// TwinCAT 3 PLC project PLC5236
// ProgramVersion: 3.1.4026.21
// libraries:
//   Tc2_EtherCAT, * (Beckhoff Automation GmbH)
//   Tc2_SerialCom, * (Beckhoff Automation GmbH)
//   Tc2_Standard, * (Beckhoff Automation GmbH)
//   Tc2_System, * (Beckhoff Automation GmbH)
//   Tc2_TcpIp, * (Beckhoff Automation GmbH)
//   Tc2_Utilities, * (Beckhoff Automation GmbH)
//   Tc3_Module, * (Beckhoff Automation GmbH)
//   VisuDialogs, * (System)
// project tree:
//   Data types/DATA_user/ USER.TcDUT, USER_ACTU.TcDUT, USER_GROUP.TcDUT
//   Data types/STRUCT COM TCPIP/ E_ClientSteps.TcDUT, E_DataExchaSteps.TcDUT, STRUCT_ClientConnect.TcDUT, STRUCT_LOG_TCPIP_CLIENT.TcDUT
//   Data types/STRUCTURE_STD/ STRUCT_JEV.TcDUT
//   Data types/ STRUCT_EVENT.TcDUT
//   Global Variables/ CONSTANT_COM_TCPIP_XTC.TcGVL, Global_Variables.TcGVL, Variable_Configuration.TcGVL
//   / PlcTask.TcTTO, Visualization Manager.TcVMO (not stored), VISU_TASK.TcTTO
//   POUs/Composant/AXES/ BLOCK_VARIATEUR_MOTEUR.TcPOU
//   POUs/Composant/ BLOCK_ACTUATOR.TcPOU, BLOCK_ACTUATOR2.TcPOU, BLOCK_VERRINE.TcPOU, MC_Reset_AX5000.TcPOU
//   POUs/Composant/EVAP/ BLOCK_CANON_ST10.TcPOU, BLOCK_IND_CREUSET_GENIUS.TcPOU, BLOCK_IND_CR_379_TELEMARK_V4.TcPOU, BLOCK_IND_CR_379_TELEMARK_V3.TcPOU, BLOCK_IND_CR_396_TELEMARK.TcPOU, BLOCK_SOURCE_GENIUS.TcPOU, BLOCK_SOURCE_JOULE.TcPOU, BLOCK_SWEEP_TELEMARK_PROG.TcPOU, BLOCK_TELEMARK_DIGITAL_SWEEP.TcPOU, BLOCK_TELEMARK_CHEETAH_SWEEP.TcPOU, BLOCK_XTAL.TcPOU, BLOCK_XTAL6.TcPOU
//   POUs/Composant/GAZ/ BLOCK_CONTROL_GAZ.TcPOU, BLOCK_MFC_ANA2.TcPOU, BLOCK_MFC_BKH.TcPOU, BLOCK_MFC_BROOKS_NoCoE.TcPOU, BLOCK_MFC_MKS_NoCoE.TcPOU
//   POUs/Composant/GENERATEURS/ ALIM_EFFLUVAGE.TcPOU
//   POUs/Composant/JAUGES/ BLOCK_BCG450_ANA.TcPOU, BLOCK_BCG450_ETHERCAT.TcPOU, BLOCK_CDG_ANA.TcPOU, BLOCK_CDG_ETHERCAT.TcPOU, BLOCK_ZX1_ANA.TcPOU
//   POUs/Composant/MVTS/ BLOCK_AXE_STD1.TcPOU, BLOCK_MOTEUR_ATV_ANA.TcPOU, BLOCK_MOTEUR_ATV_ETHERCAT.TcPOU, FB_WritePosBias.TcPOU, F_ReadMotorAbsPosition.TcPOU
//   POUs/Composant/POMPES/ BLOCK_PCR_CTI_OB.TcPOU, BLOCK_PPM.TcPOU, BLOCK_PPM_DEF.TcPOU, BLOCK_PTM_OBCV4.TcPOU, BLOCK_RS232_ONBOARD.TcPOU
//   POUs/Composant/POMPES/CRYO CTI/ BLOCK_RS232_ONBOARD_V4.TcPOU, Lecture_valeur.TcPOU
//   POUs/Composant/SERVITUDES/ BLOCK_CHILLER.TcPOU, BLOCK_CTA_HOT_COLD.TcPOU, BLOCK_SV4200.TcPOU
//   POUs/Composant/VANNES/ BLOCK_VVAT_3P.TcPOU, BLOCK_VVAT_650_ETHERCAT.TcPOU, BLOCK_VVAT_650_NO.TcPOU, BLOCK_VVAT_653_ETHERCAT.TcPOU
//   POUs/Composant/VERRINE/ BLOCK_BUZZER.TcPOU
//   POUs/FONCTION DE BASE/ ANALOG_INPUT.TcPOU, ANALOG_OUTPUT.TcPOU, BLOCK_CLIGNOTANT.TcPOU, BLOCK_CLIGNOTANT_V0_0.TcPOU, BLOCK_G7.TcPOU, BLOCK_OPERATION.TcPOU, BLOCK_RAMP.TcPOU, BLOCK_USER.TcPOU, IEEE754_INPUT.TcPOU, IEEE754_OUTPUT.TcPOU, LOG_EVENT.TcPOU, PRCDEF.TcPOU, SURVPRC.TcPOU, WRITE_CoE_BOOL.TcPOU, WRITE_CoE_WORD.TcPOU
//   POUs/FONCTION DE BASE/Format String/ FORMAT_FLOAT_STRING.TcPOU
//   POUs/Fonction/ETHER COM/ BLOCK_XTC3.TcPOU, BLOCK_XTC_CLIENT_EXCHANGE.TcPOU
//   POUs/Fonction/FONCTION EFFLUVAGE/ BLOCK_EFFLUVAGE.TcPOU
//   POUs/Fonction/FONCTION EVAPORATION/ BLOCK_EVAP.TcPOU, BLOCK_STEP_EMPILEMENT.TcPOU
//   POUs/Fonction/FONCTION MODEMARCHE/ BLOCK_1RUN_1QUARTZ.TcPOU, BLOCK_EXEC_PROC.TcPOU, BLOCK_INIT_MACHINE.TcPOU, BLOCK_MODE_MARCHE_V2_0.TcPOU, BLOCK_STEP_BOUCLE.TcPOU, BLOCK_STEP_EFFLUVAGE.TcPOU, BLOCK_STEP_TIMER.TcPOU, BLOCK_SYNCHRO_HORAIRE.TcPOU, BLOCK_USER_ACK.TcPOU
//   POUs/Fonction/FONCTION PS/ BLOCK_ROTATION_PS.TcPOU
//   POUs/Fonction/FONCTIONS COMPTEUR/ BLOCK_CPT_APP.TcPOU, BLOCK_CPT_INTEG.TcPOU, BLOCK_CPT_TEMPS.TcPOU
//   POUs/Fonction/FONCTIONS GAZ/ BLOCK_LIGNE_GAZ.TcPOU, BLOCK_LIGNE_GAZ_2_VANNES.TcPOU, BLOCK_LIGNE_GAZ_NO_DG.TcPOU, BLOCK_REGUL_PR_GAZ.TcPOU
//   POUs/Fonction/FONCTIONS MVTS/ BLOCK_ROTATION_CONTINUE_ATV.TcPOU
//   POUs/Fonction/FONCTIONS POMPAGE/ BLOCK_POMP_1E_PCR_PPM_ASS_ETHERCAT.TcPOU, BLOCK_POMP_1E_PCR_PPM_ASS_ETHERCAT_SINGER.TcPOU
//   POUs/Fonction/FONCTIONS PUISSANCE/ BLOCK_CPT_USURE.TcPOU, BLOCK_CPT_USURE_OLD.TcPOU
//   POUs/Fonction/FONCTIONS SERVITUDES/ BLOCK_LIGNE_REF.TcPOU, BLOCK_LIGNE_REF_FLOWTEMP.TcPOU, BLOCK_WREFCH1.TcPOU
//   POUs/Fonction/FONCTIONS UTILITAIRES/ CHECKSUM.TcPOU
//   POUs/Programme/ BLOCK_PRG_EFFLUVAGE.TcPOU, BLOCK_PRG_EVAP.TcPOU, BLOCK_PRG_GAZ.TcPOU, BLOCK_PRG_INFO_CLIENT.TcPOU, BLOCK_PRG_MOUVEMENT_PS.TcPOU, BLOCK_PRG_POMPAGE.TcPOU, BLOCK_PRG_SERVITUDES.TcPOU, BLOCK_PRG_VERRINE.TcPOU, MAIN.TcPOU, PRG_DEF_MANAGEMENT.TcPOU, PRG_SEC.TcPOU
//   TextLists/ GlobalTextList.TcGTLO, TextList_1Run_1Quartz.TcTLO, TextList_Actuator_Type.TcTLO, TextList_Basiques.TcTLO, TextList_Canne_Transfert.TcTLO, TextList_Chauffage.TcTLO, TextList_Config_Chauffage.TcTLO, TextList_Config_EFFLUVAGE.TcTLO, TextList_Config_Evap.TcTLO, TextList_Config_Gaz.TcTLO, TextList_Config_IAD.TcTLO, TextList_Config_Mouvements.TcTLO, TextList_Config_Pompage.TcTLO, TextList_CryoPump.TcTLO, TextList_Cryo_Relays_Parameters.TcTLO, TextList_EcoMode.TcTLO, TextList_Effluvage.TcTLO, TextList_Evap.TcTLO, TextList_Gaz.TcTLO, TextList_IAD.TcTLO, TextList_IC6.TcTLO, TextList_Infos.TcTLO, TextList_Moteurs.TcTLO, TextList_Navigation.TcTLO, TextList_Orders.TcTLO, TextList_Pompage.TcTLO, TextList_Position_Canne.TcTLO, TextList_Process.TcTLO, TextList_SA_Operations.TcTLO, TextList_Servitudes.TcTLO, TextList_STATE_Mode_Marche.TcTLO, TextList_Test_RP.TcTLO, TextList_Type_Etape.TcTLO, TextList_Type_Moteur.TcTLO, TextList_Users_Menu.TcTLO, TextList_Util_Defaut.TcTLO, TextList_Util_Group.TcTLO, TextList_Util_Userlist.TcTLO, TextList_VVAT_3P.TcTLO, TextList_VVAT_650_ETHERCAT.TcTLO
//   Visualizations/Config/Bandeaux/ VISU_BANDEAU_CFG.TcVIS
//   Visualizations/Config/CRYO/ VISU_CONFIG_REGEN.TcVIS
//   Visualizations/Config/ECOMODE/ VISU_CONFIG_ECOMODE.TcVIS
//   Visualizations/Config/EFFLUVAGE/ VISU_CONFIG_EFFLUV.TcVIS (excluded from build)
//   Visualizations/Config/EVAP/ VISU_CONFIG_EVAP.TcVIS
//   Visualizations/Config/GAZ/ VISU_CONFIG_GAZ.TcVIS
//   Visualizations/Config/MOUVEMENTS/ VISU_CONFIG_MOUVEMENTS.TcVIS
//   Visualizations/Config/POMPAGE/ VISU_CONFIG_POMPAGE.TcVIS
//   Visualizations/ MesImages.TcIPO (not stored)
//   Visualizations/Semi Auto/Elements/ SA_CACHE_ACTUATOR.TcVIS, SA_CACHE_ACTUATOR2.TcVIS, SA_EFFLUVAGE.TcVIS, SA_EVAP.TcVIS, SA_HEATING.TcVIS, SA_IAD.TcVIS, SA_LIGNE_GAZ_ANA_RAMPE.TcVIS, SA_LIGNE_GAZ_BROOKS_RAMPE.TcVIS, SA_LIGNE_GAZ_MKS_RAMPE.TcVIS, SA_POMP_1E_PCR_PPM.TcVIS, SA_POMP_1E_PCR_PPM_ASS.TcVIS, SA_POMP_1E_PCR_PPM_ASS_M11.TcVIS, SA_POMP_2E_PCR_PPM_ASS.TcVIS, SA_POMP_ENCEINTE.TcVIS, SA_POMP_SAS.TcVIS, SA_PS.TcVIS (excluded from build), SA_REGUL_GAZ.TcVIS, SA_ROT.TcVIS, SA_TEST_RP.TcVIS, SA_VERIN.TcVIS
//   Visualizations/Semi Auto/ VISU_SA.TcVIS
//   Visualizations/Symbole/CACHE/ SYM_CACHE.TcVIS, SYM_CACHE_ACTUATOR2.TcVIS
//   Visualizations/Symbole/Chauffage/ VISU_CHAUFF.TcVIS, VISU_CONFIG_CHAUFF.TcVIS, VISU_LAMPE.TcVIS
//   Visualizations/Symbole/DIVERS/ CHRONO.TcVIS
//   Visualizations/Symbole/Effluvage/ VISU_CONFIG_EFF.TcVIS, VISU_EFFLUVAGE.TcVIS
//   Visualizations/Symbole/EVAP/ VISU_ALIM_HT.TcVIS, VISU_ALIM_HT_S10.TcVIS, VISU_BAL_MANU.TcVIS, VISU_CANON.TcVIS, VISU_CANON_GENIUS_ETH.TcVIS, VISU_CANON_ST10.TcVIS, VISU_CONF_BAL.TcVIS, VISU_CONF_MAT.TcVIS, VISU_CREUSET_old.TcVIS, VISU_CREUSET.TcVIS, VISU_CREUSET_V3.TcVIS, VISU_CR_SW_GENIUS_ETH.TcVIS, VISU_HT_CANON_ST10.TcVIS, VISU_HT_GENIUS_ETH.TcVIS, VISU_SOURCE_EFFET_JOULE.TcVIS, VISU_SOURCE_EVAP_COTE_GENIUS_ETH.TcVIS, VISU_SOURCE_EVAP_COTE_ST10.TcVIS, VISU_SOURCE_EVAP_COTE_ST10_avec_emission.TcVIS, VISU_SWEEP_DIGITAL.TcVIS, VISU_SWEEP_CHEETAH.TcVIS, VISU_XTAL.TcVIS, VISU_XTAL6_ZOOM.TcVIS, VISU_XTAL6_PROD.TcVIS, VISU_XTAL_6.TcVIS
//   Visualizations/Symbole/GAZ/ VISU_CONFIG_LIGNE_GAZ_SEUIL.TcVIS, VISU_CONFIG_LIGNE_GAZ_SEUIL_MFC_MKS.TcVIS, VISU_CONFIG_LIGNE_GAZ_SURV.TcVIS, VISU_CONFIG_LIGNE_GAZ_SURV_MFC_MKS.TcVIS, VISU_CONFIG_REGUL_GAZ.TcVIS, VISU_LIGNE_GAZ.TcVIS, VISU_LIGNE_GAZ_ANA.TcVIS, VISU_LIGNE_GAZ_VGAUCHE.TcVIS, VISU_MFC_ANA.TcVIS, VISU_MFC_BROOKS.TcVIS, VISU_MFC_MKS.TcVIS
//   Visualizations/Symbole/IAD/ VISU_MARK3_PLUS.TcVIS, VISU_MARK3_PLUS_COTE.TcVIS
//   Visualizations/Symbole/JAUGES/ VISU_JAUGE_BCG450_V_HAUT.TcVIS, VISU_JAUGE_BCG450_V_HAUT_ETHERCAT.TcVIS, VISU_JAUGE_CDG045_ETHERCAT.TcVIS, VISU_JAUGE_PCG550_ETHERCAT.TcVIS
//   Visualizations/Symbole/MESURE/ VISU_IC6.TcVIS, VISU_XTC.TcVIS
//   Visualizations/Symbole/MODE_MARCHE/ VISU_BANDEAU.TcVIS, VISU_BLANCK_MANUEL.TcVIS, VISU_ECOMODE.TcVIS, VISU_ECOMODE_EVAP.TcVIS, VISU_EV_EXTRAIT.TcVIS, VISU_FCTS_SA.TcVIS, VISU_MODE_MARCHE.TcVIS
//   Visualizations/Symbole/MOUVEMENTS PS/AXE STD1/FCT_Part/ VISU_AXE_STD1_FCT_MANU.TcVIS, VISU_AXE_STD1_FCT_MANU_OSC.TcVIS, VISU_AXE_STD1_FCT_OP.TcVIS, VISU_AXE_STD1_FCT_OP_OSC.TcVIS, VISU_AXE_STD1_FCT_TRF.TcVIS, VISU_AXE_STD1_FCT_TRF_OSC.TcVIS, VISU_AXE_STD1_LIN_REL_FCT_ETAT.TcVIS, VISU_AXE_STD1_LIN_REL_FCT_ETAT_OSC.TcVIS, VISU_AXE_STD1_LIN_ROT_FCT_CONS.TcVIS, VISU_AXE_STD1_LIN_ROT_FCT_CONS_OSC.TcVIS, VISU_AXE_STD1_ROT_ABS_FCT_ETAT.TcVIS, VISU_AXE_STD1_ROT_ABS_FCT_ETAT_OSC.TcVIS
//   Visualizations/Symbole/MOUVEMENTS PS/AXE STD1/ VISU_AXE_STD1_LIN_REL.TcVIS, VISU_AXE_STD1_MANU.TcVIS, VISU_AXE_STD1_MANU_OSC.TcVIS, VISU_AXE_STD1_ROT_ABS.TcVIS, VISU_AXE_STD1_ROT_ABS_OSC.TcVIS
//   Visualizations/Symbole/MOUVEMENTS PS/ VISU_CANNE_TRANSFERT.TcVIS, VISU_CLAPET_V.TcVIS, VISU_CONFIG_POSITION_REF.TcVIS, VISU_ROT.TcVIS, VISU_VERIN_VH.TcVIS
//   Visualizations/Symbole/POMPAGE/ VISU_CONFIG_POMPAGE_CHAMBRE.TcVIS, VISU_CONFIG_POMPAGE_SAS.TcVIS, VISU_CONFIG_VANNE_ASS_VVAT650.TcVIS, VISU_CONFIG_VANNE_ASS_VVAT653_ETHERCAT.TcVIS, VISU_CONFIG_INTERJOINT.TcVIS
//   Visualizations/Symbole/POMPES/CRYO_CTI_V4/ VISU_ETAPE_REGEN.TcVIS, VISU_INFO.TcVIS, VISU_INFO_SUPP_POMPE.TcVIS, VISU_MAINT_CRYO_AC.TcVIS, VISU_MESSAGE_ALERTE.TcVIS, VISU_PARAMETRAGE_RELAY.TcVIS, VISU_POMPE_CRYO_CTI.TcVIS, VISU_RECUPERATION_ETATS.TcVIS, VISU_REGENERATION.TcVIS, VISU_TEMP_POMP_CRYO_SOLO.TcVIS
//   Visualizations/Symbole/POMPES/ VISU_POMPE_PRIMAIRE.TcVIS, VISU_POMPE_PRIMAIRE_DEF.TcVIS, VISU_POMPE_ROOTS.TcVIS, VISU_POMPE_TURBO.TcVIS, VISU_POMPE_TURBO_VPURGE.TcVIS
//   Visualizations/Symbole/PROCEDE/ VISU_INFO_PROCESS.TcVIS, VISU_MODE_QUARTZ.TcVIS
//   Visualizations/Symbole/PS/ VISU_PS.TcVIS
//   Visualizations/Symbole/SERVITUDES/ VISU_CONF_LIGNE_EAU_FLOWTEMP.TcVIS, VISU_LIGNE_EAU.TcVIS, VISU_LIGNE_EAU_NO_DEXT.TcVIS, VISU_LIGNE_EAU_FLOWTEMP.TcVIS, VISU_LIGNE_EAU_No_VE.TcVIS, VISU_TEMPRO_PLUS_90.TcVIS
//   Visualizations/Symbole/STACKER/ VISU_SUBSTRAT_NO_NUM.TcVIS
//   Visualizations/Symbole/VANNES/ VISU_VANNE_2P_H.TcVIS, VISU_VANNE_2P_H_ACT2.TcVIS, VISU_VANNE_2P_V.TcVIS, VISU_VANNE_2P_V_ACT2.TcVIS, VISU_VANNE_2P_V_NoPilot.TcVIS, VISU_VANNE_3P_H.TcVIS, VISU_VANNE_ASS_H.TcVIS, VISU_VANNE_ASS_H_MANU.TcVIS, VISU_VANNE_ASS_VAT653_ETHERCAT.TcVIS, VISU_VANNE_ASS_VAT653_ETHERCAT_MANU.TcVIS
//   Visualizations/Synoptique/ SYN_EXEC_PROC.TcVIS, SYN_INFOS.TcVIS, SYN_MANUEL.TcVIS, SYN_POMPAGE.TcVIS, SYN_PROC.TcVIS, SYN_SERVITUDES.TcVIS
//   Visualizations/Users/ UTIL_CONFIRM.TcVIS, UTIL_DEFAUT.TcVIS, UTIL_DELOG.TcVIS, UTIL_GROUP.TcVIS, UTIL_LOG.TcVIS, UTIL_MENU.TcVIS, UTIL_MOD_GROUP.TcVIS, UTIL_MOD_USER.TcVIS, UTIL_NEW_GROUP.TcVIS, UTIL_NEW_USER.TcVIS, UTIL_OPT.TcVIS, UTIL_USER.TcVIS
// real-time tasks:
//   TASK PlcTask: cycle T#10ms, priority 20, ADS port 350
//   TASK VISU_TASK: cycle T#200000us, priority 30, ADS port 351
// I/O:
//   DEVICE PC1 (EtherCAT) (disabled), AmsNetId 172.18.237.251.2.1
//     IMX1 (EK1100) [EK1100 EtherCAT Coupler (2A E-Bus)]
//       X1.0 (EL6070) [EL6070 1Ch. Licensing-Terminal]
//       X1.1 (EL1008) [EL1008 8Ch. Dig. Input 24V, 3ms]
//       X1.2 (EL1008) [EL1008 8Ch. Dig. Input 24V, 3ms]
//       X1.3 (EL1008) [EL1008 8Ch. Dig. Input 24V, 3ms]
//       X1.4 (EL1008) [EL1008 8Ch. Dig. Input 24V, 3ms]
//       X1.5 (EL3104) [EL3104 4Ch. Ana. Input +/-10V Diff.] (disabled)
//       X1.5 (EL3064) [EL3064 4Ch. Ana. Input 0-10V]
//       X1.6 (EL4004) [EL4004 4Ch. Ana. Output 0-10V, 12bit]
//       X1.7 (EL2008) [EL2008 8Ch. Dig. Output 24V, 0.5A]
//       X1.11 (EL2008) [EL2008 8Ch. Dig. Output 24V, 0.5A]
//       X1.12 (EL2008) [EL2008 8Ch. Dig. Output 24V, 0.5A]
//       X1.13 (EL2624) [EL2624 4Ch. Relay Output, NO (125V AC / 30V DC)]
//       X1.14 (EL2624) [EL2624 4Ch. Relay Output, NO (125V AC / 30V DC)]
//       X1.15 (EL2624) [EL2624 4Ch. Relay Output, NO (125V AC / 30V DC)]
//       X1.16 (EL2624) [EL2624 4Ch. Relay Output, NO (125V AC / 30V DC)]
//       X1.17 (EL9011) [EL9011 End Terminal]
//     VRPS (ATV320 EtherCAT) [ATV320 EtherCAT]
//     IMX2 (EK1100) [EK1100 EtherCAT Coupler (2A E-Bus)]
//       X2.1 (EL1008) [EL1008 8Ch. Dig. Input 24V, 3ms]
//       X2.2 (EL1008) [EL1008 8Ch. Dig. Input 24V, 3ms]
//       X2.3 (EL6224) [EL6224 (IO Link Master)]
//       X2.4 (EL6224) [EL6224 (IO Link Master)]
//       X2.11 (EL2008) [EL2008 8Ch. Dig. Output 24V, 0.5A]
//       X2.12 (EL2008) [EL2008 8Ch. Dig. Output 24V, 0.5A]
//       X2.13 (EL2624) [EL2624 4Ch. Relay Output, NO (125V AC / 30V DC)]
//       X2.14 (EL2624) [EL2624 4Ch. Relay Output, NO (125V AC / 30V DC)]
//       X2.14 (EL9011) [EL9011 End Terminal]
//     DG11 (G Series MFC) [G Series EtherCAT MFC]
//     DG12 (G Series MFC) [G Series EtherCAT MFC]
//     VS11 (VAT valve S653) [VAT valve S653]
//     M11 (BCG 450) [ BCG 450 V1.3.0.0 ]
//     M11 (BCG 450 V 1.3.0.0) [BCG 450 V 1.3.0.0] (disabled)
//   DEVICE COM_Cryos (COM Port RS232) (disabled)
// variable links:
//   PLC5236/PLC5236 Instance <-> COM_Cryos (COM Port RS232)
//     PlcTask Inputs/.PRG_POMPAGE.COM_CRYOS.IN_COM/D[{0..63}] <-> Inputs/Data{1..64}  (64 links)
//     PlcTask Inputs/.PRG_POMPAGE.COM_CRYOS.IN_COM/SerStatus <-> Inputs/Status
//     PlcTask Outputs/.PRG_POMPAGE.COM_CRYOS.OUT_Com/D[{0..63}] <-> Outputs/Data{1..64}  (64 links)
//     PlcTask Outputs/.PRG_POMPAGE.COM_CRYOS.OUT_Com/SerCtrl <-> Outputs/Ctrl
//   PLC5236/PLC5236 Instance <-> PC1 (EtherCAT)/DG11 (G Series MFC)
//     PlcTask Inputs/.PRG_GAZ.DG[1].IN_Measure <-> Inputs ( Default)/Flow Reading
//     PlcTask Outputs/.PRG_GAZ.DG[1].OUT_Setpoint <-> Outputs (Default)/Flow SP
//   PLC5236/PLC5236 Instance <-> PC1 (EtherCAT)/DG12 (G Series MFC)
//     PlcTask Inputs/.PRG_GAZ.DG[2].IN_Measure <-> Inputs ( Default)/Flow Reading
//     PlcTask Outputs/.PRG_GAZ.DG[2].OUT_Setpoint <-> Outputs (Default)/Flow SP
//   PLC5236/PLC5236 Instance <-> PC1 (EtherCAT)/IMX1 (EK1100)/X1.1 (EL1008)
//     PlcTask Inputs/.PRG_EVAP.SOURCE1.IN_HV_OK <-> Channel 7/HVOK
//     PlcTask Inputs/.PRG_EVAP.SOURCE1.IN_HV_ON <-> Channel 8/HVON
//     PlcTask Inputs/.PRG_MOUVEMENT_PS.IN_JOG <-> Channel 6/S-JOG
//     PlcTask Inputs/.PRG_POMPAGE.IN_FE11T <-> Channel 2/FE11T
//     PlcTask Inputs/.PRG_POMPAGE.IN_PP11M <-> Channel 3/PP11M
//     PlcTask Inputs/.PRG_POMPAGE.IN_PR11M <-> Channel 4/PR11M
//     PlcTask Inputs/.PRG_POMPAGE.IN_PS11M <-> Channel 5/PS11M
//     PlcTask Inputs/MAIN.IN_MM1_Brut <-> Channel 1/M11
//     PlcTask Inputs/MAIN.In_Data_INValid <-> WcState/WcState
//   PLC5236/PLC5236 Instance <-> PC1 (EtherCAT)/IMX1 (EK1100)/X1.11 (EL2008)
//     PlcTask Outputs/.PRG_EVAP.OUT_MEG1 <-> Channel 5/MAEG1
//     PlcTask Outputs/.PRG_EVAP.OUT_MPR230 <-> Channel 1/MECO
//     PlcTask Outputs/.PRG_POMPAGE.OUT_PP11 <-> Channel 2/PP11
//     PlcTask Outputs/.PRG_POMPAGE.OUT_PR11 <-> Channel 3/PR11
//     PlcTask Outputs/.PRG_POMPAGE.OUT_PS11 <-> Channel 4/PS11
//   PLC5236/PLC5236 Instance <-> PC1 (EtherCAT)/IMX1 (EK1100)/X1.12 (EL2008)
//     PlcTask Outputs/.PRG_EVAP.OUT_CR{11..14} <-> Channel {1..4}/CR{11..14}  (4 links)
//     PlcTask Outputs/.PRG_EVAP.OUT_CR_RMT <-> Channel 5/CR_RMT
//   PLC5236/PLC5236 Instance <-> PC1 (EtherCAT)/IMX1 (EK1100)/X1.13 (EL2624)
//     PlcTask Outputs/.PRG_EVAP.SOURCE1.OUT_HV <-> Channel 1/MHV
//     PlcTask Outputs/.PRG_EVAP.SOURCE1.OUT_ITLCK_HVAC <-> Channel 4/HVAC
//     PlcTask Outputs/.PRG_EVAP.SOURCE1.OUT_ITLCK_VAC <-> Channel 3/VAC
//     PlcTask Outputs/.PRG_EVAP.SOURCE1.OUT_SRC <-> Channel 2/MFIL
//   PLC5236/PLC5236 Instance <-> PC1 (EtherCAT)/IMX1 (EK1100)/X1.14 (EL2624)
//     PlcTask Outputs/.PRG_EVAP.OUT_MEJ1 <-> Channel 3/MEJ1
//     PlcTask Outputs/.PRG_EVAP.OUT_MEJ2 <-> Channel 4/MEJ2
//     PlcTask Outputs/.PRG_EVAP.SOURCE1.OUT_ITLCK_WAT <-> Channel 1/WAT
//   PLC5236/PLC5236 Instance <-> PC1 (EtherCAT)/IMX1 (EK1100)/X1.15 (EL2624)
//     PlcTask Outputs/.PRG_EVAP.OUT_SWB1 <-> Channel 2/SWB1
//     PlcTask Outputs/.PRG_EVAP.OUT_SWB2 <-> Channel 3/SWB2
//     PlcTask Outputs/.PRG_EVAP.OUT_SWB3 <-> Channel 4/SWB3
//   PLC5236/PLC5236 Instance <-> PC1 (EtherCAT)/IMX1 (EK1100)/X1.16 (EL2624)
//     PlcTask Outputs/.PRG_EVAP.OUT_SWB4 <-> Channel 1/SWB4
//     PlcTask Outputs/.PRG_EVAP.OUT_SW_RMT <-> Channel 3/SW_RMT
//   PLC5236/PLC5236 Instance <-> PC1 (EtherCAT)/IMX1 (EK1100)/X1.2 (EL1008)
//     PlcTask Inputs/.PRG_EVAP.IN_CR{11..14}T <-> Channel {2..5}/CR{11..14}T  (4 links)
//     PlcTask Inputs/.PRG_EVAP.SOURCE1.IN_SRC_ON <-> Channel 1/FILON
//   PLC5236/PLC5236 Instance <-> PC1 (EtherCAT)/IMX1 (EK1100)/X1.3 (EL1008)
//     PlcTask Inputs/.PRG_EVAP.XTC3.IN_CD{31..36}T <-> Channel {2..7}/CD{11..16}T  (6 links)
//     PlcTask Inputs/MAIN.IN_MA1T <-> Channel 8/MA1T
//   PLC5236/PLC5236 Instance <-> PC1 (EtherCAT)/IMX1 (EK1100)/X1.4 (EL1008)
//     PlcTask Inputs/.PRG_EVAP.IN_SW_RDY <-> Channel 3/SW-RDY
//     PlcTask Inputs/.PRG_EVAP.IN_SW_REM <-> Channel 1/SW-RMT
//     PlcTask Inputs/.PRG_EVAP.IN_SW_RUN <-> Channel 2/SW-RUN
//   PLC5236/PLC5236 Instance <-> PC1 (EtherCAT)/IMX1 (EK1100)/X1.5 (EL3064)
//     PlcTask Inputs/.PRG_EVAP.SOURCE1.IN_FILQ <-> AI Standard Channel 3/FILQ
//     PlcTask Inputs/.PRG_EVAP.SOURCE1.IN_IEMQ <-> AI Standard Channel 2/IEMQ
//     PlcTask Inputs/.PRG_EVAP.SOURCE1.IN_UHVQ <-> AI Standard Channel 1/HVQ
//   PLC5236/PLC5236 Instance <-> PC1 (EtherCAT)/IMX1 (EK1100)/X1.6 (EL4004)
//     PlcTask Outputs/.PRG_EVAP.SOURCE1.OUT_QIEM <-> AO Outputs Channel 2/QFIL
//     PlcTask Outputs/.PRG_EVAP.SOURCE1.OUT_QUHV <-> AO Outputs Channel 1/QHV
//   PLC5236/PLC5236 Instance <-> PC1 (EtherCAT)/IMX1 (EK1100)/X1.7 (EL2008)
//     PlcTask Outputs/.PRG_VERRINE.OUT_Orange <-> Channel 2/VER1-O
//     PlcTask Outputs/.PRG_VERRINE.OUT_Rouge <-> Channel 3/VER1-R
//     PlcTask Outputs/.PRG_VERRINE.OUT_Vert <-> Channel 1/VER1-V
//   PLC5236/PLC5236 Instance <-> PC1 (EtherCAT)/IMX2 (EK1100)/X2.1 (EL1008)
//     PlcTask Inputs/.PRG_EVAP.QZ1.QZ{11..14}T <-> Channel {5..8}/QZ{11..14}T  (4 links)
//     PlcTask Inputs/.PRG_POMPAGE.IN_ST11 <-> Channel 1/ST111
//     PlcTask Inputs/.PRG_POMPAGE.IN_ST12 <-> Channel 2/ST112
//   PLC5236/PLC5236 Instance <-> PC1 (EtherCAT)/IMX2 (EK1100)/X2.11 (EL2008)
//     PlcTask Outputs/.PRG_EVAP.QZ1.OUT_QZ1 <-> Channel 5/QZ1
//     PlcTask Outputs/.PRG_GAZ.OUT_VG11 <-> Channel 6/VG11
//     PlcTask Outputs/.PRG_GAZ.OUT_VG12 <-> Channel 7/VG12
//     PlcTask Outputs/.PRG_POMPAGE.OUT_VH11 <-> Channel 4/VH11
//     PlcTask Outputs/.PRG_POMPAGE.OUT_VINT <-> Channel 3/VINT
//     PlcTask Outputs/.PRG_POMPAGE.OUT_VN2PP11 <-> Channel 8/VN2PP11
//   PLC5236/PLC5236 Instance <-> PC1 (EtherCAT)/IMX2 (EK1100)/X2.12 (EL2008)
//     PlcTask Outputs/.PRG_SERVITUDES.OUT_VE{1..5} <-> Channel {1..5}/VE{1..5}  (5 links)
//   PLC5236/PLC5236 Instance <-> PC1 (EtherCAT)/IMX2 (EK1100)/X2.13 (EL2624)
//     PlcTask Outputs/.PRG_EVAP.OUT_ICC11 <-> Channel 2/ICCEG1
//     PlcTask Outputs/.PRG_EVAP.OUT_ICC12 <-> Channel 4/ICCEJ1
//     PlcTask Outputs/.PRG_EVAP.OUT_OCC11 <-> Channel 1/OCCEG1
//     PlcTask Outputs/.PRG_EVAP.OUT_OCC12 <-> Channel 3/OCCEJ1
//   PLC5236/PLC5236 Instance <-> PC1 (EtherCAT)/IMX2 (EK1100)/X2.14 (EL2624)
//     PlcTask Outputs/.PRG_EVAP.OUT_ICC13 <-> Channel 2/ICCEJ2
//     PlcTask Outputs/.PRG_EVAP.OUT_OCC13 <-> Channel 1/OCCEJ2
//   PLC5236/PLC5236 Instance <-> PC1 (EtherCAT)/IMX2 (EK1100)/X2.2 (EL1008)
//     PlcTask Inputs/.PRG_EVAP.QZ1.QZ15T <-> Channel 1/QZ15T
//     PlcTask Inputs/.PRG_EVAP.QZ1.QZ16T <-> Channel 2/QZ16T
//   PLC5236/PLC5236 Instance <-> PC1 (EtherCAT)/M11 (BCG 450)
//     PlcTask Inputs/.PRG_POMPAGE.IN_M11Q <-> Transmit PDO Mapping Module 1/Combination Gauge Active Value
//     PlcTask Inputs/.PRG_POMPAGE.M11.IN_Active_Sensor <-> Transmit PDO Mapping Module 1/Combination Gauge Active Sensor Number
//     PlcTask Inputs/.PRG_POMPAGE.M11.IN_WcState <-> WcState/WcState
//   PLC5236/PLC5236 Instance <-> PC1 (EtherCAT)/VRPS (ATV320 EtherCAT)
//     PlcTask Outputs/.PRG_MOUVEMENT_PS.ROTATION_PS.PS.OUT_Velocity <-> Outputs/Target Velocity

CONFIGURATION PLC5236
    RESOURCE PLC ON TwinCAT3
        TASK PlcTask(INTERVAL := T#10ms, PRIORITY := 20);
        TASK VISU_TASK(INTERVAL := T#200000us, PRIORITY := 30);
        PROGRAM MAIN WITH PlcTask : MAIN;
        PROGRAM VisuElems_Visu_Prg WITH VISU_TASK : VisuElems.Visu_Prg;
    END_RESOURCE
END_CONFIGURATION

// ---- Data types/DATA_user/USER.TcDUT
TYPE USER :

STRUCT

	LOGIN:			STRING[30];
	PASS:			STRING[30];
	PASS_DISPLAY:	STRING[30];
	NOM:			STRING[30];
	PRENOM:			STRING[30];
	GROUPE:			STRING[30];

END_STRUCT

END_TYPE

// ---- Data types/DATA_user/USER_ACTU.TcDUT
TYPE USER_ACTU :
STRUCT
	LOGIN:					STRING[30];
	PASS:					STRING[30];
	NOM:					STRING[30];
	PRENOM:				STRING[30];
	GROUPE:				STRING[30];
	PROGRAMMATION:		BOOL;			(*Edition de procédé*)
	MAINTENANCE:			BOOL;			(*Passage en mode maintenance, consignation, journal des évènements*)
	SUPERVISEUR:			BOOL;
	PRODUCTION:			BOOL;			(*Passage en production, arrêt production, interruption/reprise procédé, arrêt procédé, pause procédé*)
	CONF_MACHINE:			BOOL;			(*Configuration machine hors motorisation transfert*)
	FONCTION_SA:			BOOL;			(*Fonctions avancées hors production*)
	CONF_TRF:				BOOL;			(*Configuration machine spécifique motorisation transfert*)
	MODIF_ENLIGNE:			BOOL;			(*Rechargement, passage étape suivante, modification consignes sa en production*)
	ARCHIVE_EV:			BOOL;			(*Gestion du journal des évènements, TR'AC*)
	DECONSIGNATION:		BOOL;			(*Déconsignation module*)
END_STRUCT
END_TYPE

// ---- Data types/DATA_user/USER_GROUP.TcDUT
TYPE USER_GROUP :

STRUCT

	NOM:					STRING[30];
	PROGRAMMATION:		BOOL;
	MAINTENANCE:			BOOL;
	SUPERVISEUR:			BOOL;
	PRODUCTION:			BOOL;
	CONF_MACHINE:			BOOL;
	FONCTION_SA:			BOOL;
	CONF_TRF:				BOOL;			(*Configuration machine spécifique motorisation transfert*)
	MODIF_ENLIGNE:			BOOL;			(*Rechargement, passage étape suivante, modification consignes sa en production*)
	ARCHIVE_EV:			BOOL;			(*Gestion du journal des évènements, TR'AC*)
	DECONSIGNATION:		BOOL;			(*Déconsignation module*)
END_STRUCT

END_TYPE

// ---- Data types/STRUCT COM TCPIP/E_ClientSteps.TcDUT
TYPE E_ClientSteps :
(
	CLIENT_STATE_IDLE,
	CLIENT_STATE_CONNECT_START,
	CLIENT_STATE_CONNECT_WAIT,
	CLIENT_STATE_DATAEXCHA_START,
	CLIENT_STATE_DATAEXCHA_WAIT,
	CLIENT_STATE_CLOSE_START,
	CLIENT_STATE_CLOSE_WAIT,
	CLIENT_STATE_ERROR,
	CLIENT_STATE_DATA_ANALYSE
);
END_TYPE

// ---- Data types/STRUCT COM TCPIP/E_DataExchaSteps.TcDUT
TYPE E_DataExchaSteps :
(
	DATAEXCHA_STATE_IDLE,
	DATAEXCHA_STATE_SEND_START,
	DATAEXCHA_STATE_SEND_WAIT,
	DATAEXCHA_STATE_RECEIVE_START,
	DATAEXCHA_STATE_RECEIVE_WAIT,
	DATAEXCHA_STATE_ERROR,
	DATAEXCHA_STATE_RECEIVE_BEFORE_RETRY_START,
	DATAEXCHA_STATE_RECEIVE_BEFORE_RETRY_WAIT
);
END_TYPE

// ---- Data types/STRUCT COM TCPIP/STRUCT_ClientConnect.TcDUT
(*structure de variable associée à la gestion d'un client TCPIP*)
TYPE STRUCT_ClientConnect :
STRUCT
	fbConnectTON:		TON;	(*temporisation de reconnexion sur le client*)
	fbDataExchaTON:		TON;		(*temporisation cyclique de requête sur le client*)
	eStep:				E_ClientSteps;	(*Etat de la séquence de gestion du client*)
	bBusy:				BOOL;	(*indicateur de gestion du client*)
	bError:				BOOL;	(*indicateur d'erreur*)
	nErrid:				UDINT;	(*N° d'erreur*)
	ErrDescription		: T_MAXSTRING;
	bEnable				:BOOL;	(*autorisation de lecture cyclique des paramètres*)
	bConnected:			BOOL;	(*etat de connexion*)
	nStepInError:			UDINT;	(*N° d'étape en erreur*)
	nRequest:			UINT;	(*N° de requete à envoyer*)
	fbConnect			: FB_SocketConnect := ( sSrvNetId := ''  );
	fbClose				: FB_SocketClose := ( sSrvNetId := '', tTimeout := DEFAULT_ADS_TIMEOUT );
	fbClientDataExcha		: BLOCK_XTC_CLIENT_EXCHANGE;
	hSocket				: T_HSOCKET;
	ConnectTime			: TIME;	(*Valeur de la temporisation avant reconnexion du port*)
	ExchangeCycleTime	: TIME;	(*Valeur de temporisation d'échange*)
	Compteur_connection	: UDINT;
END_STRUCT
END_TYPE

// ---- Data types/STRUCT COM TCPIP/STRUCT_LOG_TCPIP_CLIENT.TcDUT
(*Structure du journal d'émission / réception*)
TYPE STRUCT_LOG_TCPIP_CLIENT :
STRUCT
	RX				: ARRAY[0..MAX_RXBUFFER_SIZE] OF BYTE; 		(*Stockage des répondes du buffer*)
	TX				: ARRAY[0..MAX_TXBUFFER_SIZE] OF BYTE; 		(*Stockage des répondes du buffer*)
	ERR			: T_MAXSTRING;
END_STRUCT
END_TYPE

// ---- Data types/STRUCTURE_STD/STRUCT_JEV.TcDUT
TYPE STRUCT_JEV :
STRUCT
	STATE_dt:		DT;
	STATE_App:		STRING;
	STATE_Path:		STRING;
	STATE_Title:	STRING(200);
END_STRUCT
END_TYPE

// ---- Data types/STRUCT_EVENT.TcDUT
TYPE STRUCT_EVENT :
STRUCT
	_ID:				UINT;
	_VAL1:			STRING;
	_VAL2:			STRING;
	_VAL3:			STRING;
	_HORODAT:		DT;
	_MS:			UINT;
	_TYPE:			BOOL;	(*True = apparition, False=disparition*)
END_STRUCT
END_TYPE

// ---- Global Variables/CONSTANT_COM_TCPIP_XTC.TcGVL
{attribute 'Tc2GvlVarNames'}

VAR_GLOBAL CONSTANT
	{attribute 'OPC.UA.DA'  := '1'}
	MAX_BUFFER_DIALOG							: UDINT := 100;	(*Taille max du buffer de mémorisation des trames d'émission-réception*)
	{attribute 'OPC.UA.DA'  := '1'}
	MAX_RXBUFFER_SIZE							: UDINT := 1000;    	(*Taille max du buffer de réception*)
	{attribute 'OPC.UA.DA'  := '1'}
	MAX_TXBUFFER_SIZE							: UDINT := 255;    	(*Taille max du buffer d'émission*)
	(* Codes d'erreur spécifiques *)
	{attribute 'OPC.UA.DA'  := '1'}
	ERROR_RECEIVE_BUFFER_OVERFLOW				: UDINT := 16#8101; (* receive buffer overflow*)
	{attribute 'OPC.UA.DA'  := '1'}
	ERROR_RECEIVE_TIMEOUT						: UDINT := 16#8102; (* receive timeout error *)
	{attribute 'OPC.UA.DA'  := '1'}
	ERROR_MESSAGE_CCB							: UDINT := 16#8103; (*bad CCB*)
	{attribute 'OPC.UA.DA'  := '1'}
	ERROR_MESSAGE_LENGTH						: UDINT := 16#8104; (*Bad message length*)
	{attribute 'OPC.UA.DA'  := '1'}
	ERROR_MISSING_ACK							: UDINT := 16#8105; (*ACK missing*)
END_VAR

// ---- Global Variables/Global_Variables.TcGVL
{attribute 'Tc2GvlVarNames'}
VAR_GLOBAL

	(*Variable de vérification de chargement des variables persistentes ok*)
	{attribute 'OPC.UA.DA'  := '1'}
	STATE_Charg_Persistentes_Ok:	BOOL;

	(*Général*)
	{attribute 'OPC.UA.DA'  := '1'}
	MACHINE:						BLOCK_MODE_MARCHE_V2_0;
	{attribute 'OPC.UA.DA'  := '1'}
	INIT_MACHINE:					BLOCK_INIT_MACHINE;
	{attribute 'OPC.UA.DA'  := '1'}
	EXECPROC:						BLOCK_EXEC_PROC;
	{attribute 'OPC.UA.DA'  := '1'}
	MODE_QUARTZ_PROD:				BLOCK_1RUN_1QUARTZ;

	(*Instances des PRG*)
	{attribute 'OPC.UA.DA'  := '1'}
	PRG_USER:						BLOCK_USER;
	{attribute 'OPC.UA.DA'  := '1'}
	PRG_EFFLUVAGE:					BLOCK_PRG_EFFLUVAGE;
	{attribute 'OPC.UA.DA'  := '1'}
	PRG_EVAP:						BLOCK_PRG_EVAP;
	{attribute 'OPC.UA.DA'  := '1'}
	PRG_MOUVEMENT_PS:				BLOCK_PRG_MOUVEMENT_PS;
	{attribute 'OPC.UA.DA'  := '1'}
	PRG_POMPAGE:					BLOCK_PRG_POMPAGE;
	{attribute 'OPC.UA.DA'  := '1'}
	PRG_SERVITUDES:					BLOCK_PRG_SERVITUDES;
	{attribute 'OPC.UA.DA'  := '1'}
	PRG_GAZ:						BLOCK_PRG_GAZ;
	{attribute 'OPC.UA.DA'  := '1'}
	PRG_VERRINE:					BLOCK_PRG_VERRINE;
	{attribute 'OPC.UA.DA'  := '1'}
	PRG_INFO_CLIENT:				BLOCK_PRG_INFO_CLIENT;

	(*Securisation du mode manuel*)
	{attribute 'OPC.UA.DA'  := '1'}
	STATE_PROGRESS_BAR_MANU: 		USINT;
	{attribute 'OPC.UA.DA'  := '1'}
	TIMER_SECU_OFF:					TON;
	{attribute 'OPC.UA.DA'  := '1'}
	IHM_SHUNT_SECU:					BOOL;		(*apui sur bouton de shunt des sécu*)
	{attribute 'OPC.UA.DA'  := '1'}
	IHM_SECU_ON:					BOOL;		(*appui sur bouton de reprise du mode manu securisé*)


	(*variable générale de securités désactivées*)
	{attribute 'OPC.UA.DA'  := '1'}
	MANUAL_SAFETY_OFF:				BOOL;		(* ~ (OPC : 1 : available for OPC-clients) *)

	(*variables liées à la gestion des paramètres persistents*)
	{attribute 'OPC.UA.DA'  := '1'}
	RQ_PARAM_SYSTEM:				BOOL;
	{attribute 'OPC.UA.DA'  := '1'}
	PARAM_SYSTEM_OK:				BOOL;		(*drapeau indiquant que le paramètrage du système est OK*)
	{attribute 'OPC.UA.DA'  := '1'}
	RQ_SAV_PERSISTENT:				BOOL;		(*Demande de sauvegarde des variables persistants*)


	(*Variables de navigation*)
	{attribute 'OPC.UA.DA'  := '1'}
	SHOW_SM_SA:					BOOL;
	{attribute 'OPC.UA.DA'  := '1'}
	SHOW_CONFIRM_REGEN:			BOOL;
	{attribute 'OPC.UA.DA'  := '1'}
	SHOW_MODIF_RAMPE:			BOOL;
	{attribute 'OPC.UA.DA'  := '1'}
	VISU_INDEX_MANU:			USINT;

	DEBUG_BOOL1:	BOOL;
	DEBUG_BOOL2: 	BOOL;
	DEBUG_BOOL3:	BOOL;
	DEBUG_BOOL4:	BOOL;
	DEBUG_BOOL5:	BOOL;
	DEBUG_BOOL6:	BOOL;
	DEBUG_BOOL7:	BOOL;
	DEBUG_BOOL8:	BOOL;
	DEBUG_BOOL9:	BOOL;
	DEBUG_BOOL10:	BOOL;
	DEBUG_BOOL11:	BOOL;
	DEBUG_BOOL12:	BOOL;
	DEBUG_REAL1:	REAL;
	DEBUG_REAL2:	REAL;
	VAR_Mem_ECO:	BOOL;
	
END_VAR

// ---- Global Variables/Variable_Configuration.TcGVL
{attribute 'Tc2GvlVarNames'}
VAR_CONFIG
END_VAR

// ---- POUs/Programme/MAIN.TcPOU
PROGRAM MAIN
VAR
	VAR_FB_WritePersistentData:		FB_WritePersistentData;
	FM_BUSY:						R_TRIG;
	FM_ERROR:						R_TRIG;
	FM_PCSY:						R_TRIG;
	BIT_1s:							BLOCK_CLIGNOTANT;
	STEP_USER_ACK:					BLOCK_USER_ACK;				(*Block validation opérateur*)
	STEP_SYNHRO_HORAIRE:			BLOCK_SYNCHRO_HORAIRE;
	STEP_TIMER:						BLOCK_STEP_TIMER;
	STEP_EFFLUVAGE:					BLOCK_STEP_EFFLUVAGE;
	STEP_EMPILEMENT:				BLOCK_STEP_EMPILEMENT;
	STEP_BOUCLE:					BLOCK_STEP_BOUCLE;

	IN_MM1_Brut	AT%I*:				BOOL;
	IN_MM1:							BOOL;
	IN_PT1	AT%I*:					BOOL;
	IN_MA1T	AT%I*:					BOOL;
	IN_MA2T	AT%I*:					BOOL;
	In_Data_INValid	AT%I*:			BOOL;

	Process:			NT_StartProcess;
	bStartVerif:		BOOL;		(*Démarrage du laucnher*)
	bTest:				BOOL;		(*Booléen pour test lecture*)

	(*Fonction de calcul d'usure*)
	CPT_USURE:		BLOCK_CPT_USURE;
	
	VAR_Invisible_Delog:			BOOL;
	
	(*Tr'AC variables*)
	PING_TRAC:			BOOL;
	TRAC_PW:			STRING:='Ac_74960';
	TRAC_SLOW_RECORD: 	BOOL;
	TRAC_EXPORT_AUTO:	BOOL;
	TRAC_RECORD:		BOOL;
	TRAC_PROCESS_NAME: 	STRING;
	Enr_TRAC:			BOOL;
	
	(*ACSoft variables*)
	PING_ACSOFT:		BOOL;
	
	(*Variables EcoMode*)
	TIMER_Inactivite:					TON;
	
	VAR_Debug_Bool:		BOOL;
	I_STOP_ROTATION_OK: INT;
	CO_Stop: INT;
END_VAR

VAR_INPUT PERSISTENT
END_VAR

(*IN MM1 récupéré avec data valid de X1.1*)
IN_MM1 := IN_MM1_Brut;// AND NOT In_Data_INValid;
VAR_Debug_Bool	:=	In_Data_INValid;

(*Vérification du chargement ok des persistentes :
bit 4 à 1 pour wbp chargé correctement, et bit 5 à 0 pour fichier backup pas chargé (possibilité de variables erronées dans ce cas)*)
(*STATE_Charg_Persistentes_Ok	:=	SystemInfo.bootDataFlags.4 AND NOT SystemInfo.bootDataFlags.5;*)

STATE_Charg_Persistentes_Ok := TRUE;

(*Parametres statiques*)
MACHINE.IdParent				:=		'RACINE';
MACHINE.MNEMO					:=		'MACHINE';
MACHINE.IdXML					:=		'0';
MACHINE.TagXML					:=		0;

MACHINE.CONF_No_MA1T 			:= 		FALSE;
MACHINE.CONF_No_MA2T 			:= 		TRUE;

MACHINE.CONF_Model				:= 		'AC3000 EVA 900';
MACHINE.CONF_Name 				:=		'EVA 900 N°1';
MACHINE.CONF_Affaire			:=		'5236';
MACHINE.CONF_Author				:=  	'LDS';
MACHINE.CONF_Customer			:=		'SINGER';
MACHINE.CONF_SerialNumber		:=		'M02-23/441';
MACHINE.CONF_Version			:=		'0.0';
MACHINE.CONF_VerDate			:=		'09/2026';

MACHINE.CONF_TrAC				:=	TRUE;
MACHINE.CONF_ACSoft				:=	TRUE;

MODE_QUARTZ_PROD.CONF_N_Quartz_total	:=	6;
MODE_QUARTZ_PROD.CONF_N_Quartz_secours	:=	1;

(*gestion de la sauvegarde des paramètres persistents : on fait retomber l'état param_system_ok*)
IF RQ_PARAM_SYSTEM THEN
 	PARAM_SYSTEM_OK	 := FALSE;
END_IF

MACHINE(
	IN_PT1:= 				TRUE,
	IN_MM1:= 				IN_MM1,
	IN_MA1T:= 				IN_MA1T,
	IN_MA2T:= 				TRUE,
	EN_Auto:= 				STATE_Charg_Persistentes_Ok,
	EN_Manu:= 				TRUE,
	EN_Prod:= 				PRG_POMPAGE.DOOR
							AND PRG_EVAP.QZ1.OP_Positionnement.AR
							AND PRG_EVAP.QZ1.OP_Scan_Quartz.AR,
	EN_Inter_Prod:= 		TRUE,
	EN_Reprise_Prod:= 		TRUE,
	EN_Standby:=			TRUE,
	I_Init_OK:= 			INIT_MACHINE.STATE_OK,
	I_Prep_Prod_OK:= 		INIT_MACHINE.STATE_OK,
	I_PROCEDE_ok:= 			EXECPROC.STATE_OK,
	I_ARRET_PROCEDE_OK:= 	INIT_MACHINE.STATE_OK,
	I_INTER_PROD_OK:=  		INIT_MACHINE.STATE_OK,
	I_MOTEUR_INTER_OK:=		EXECPROC.STATE_INTERRUPTED,
	I_def_stop:= 			EXECPROC.DEF_PROCESS_LOADING.DEF
							OR PRG_POMPAGE.POMPAGE.OP_Isolement.DEF_AUTO_ON.DEF,
	I_def_inter:=			EXECPROC.DEF_READ_STEP.DEF
							OR EXECPROC.DEF_STEP_REJECTED.DEF
							OR STEP_EMPILEMENT.DEF_READ_LAYER.DEF
							OR STEP_EMPILEMENT.DEF_READ_LAYER_ANT.DEF
							OR STEP_EMPILEMENT.DEF_PROG_QZ.DEF
							OR STEP_EMPILEMENT.DEF_RAZ_QZ.DEF
							OR (STEP_EMPILEMENT.DEF_QF.DEF AND NOT MODE_QUARTZ_PROD.STATE_Mode)
							OR STEP_EMPILEMENT.DEF_CONTROLLER_STOPPED.DEF
							OR STEP_EFFLUVAGE.DEF_SEUIL_POMPAGE_PRIM.DEF
							OR STEP_EFFLUVAGE.DEF_SEUIL_VIDE_EFFLUVAGE.DEF
							OR PRG_EVAP.STATE_Def_IProc
							OR PRG_GAZ.STATE_Def_IProc
							OR PRG_POMPAGE.STATE_Def_IProc
							OR PRG_EFFLUVAGE.STATE_Def_IProc
							OR PRG_MOUVEMENT_PS.STATE_Def_IProc
							OR MODE_QUARTZ_PROD.DEF_Stop_Quartz.DEF OR MODE_QUARTZ_PROD.DEF_No_Quartz.DEF
							OR MACHINE.DEF_Air.DEF,
	I_PROCEDE_WD_Ar:=		TRUE,
	I_PROCEDE_WD_Ok:=		EXECPROC.STATE_OK,
	I_Standby_Ok:=			NOT PRG_EVAP.OUT_MEG1 AND NOT PRG_EVAP.OUT_MPR230,
	I_WakeUp_Ok:= 			PRG_EVAP.XTC3.STATE_READY,
	PING_ACSoft:=			PING_ACSOFT,
	PING_TRAC:=				PING_TRAC);


INIT_MACHINE(
	I_STOP_EVAP_OK := PRG_EVAP.EVAPS1.OP_Stop.OK AND PRG_EVAP.EVAPS2.OP_Stop.OK AND PRG_EVAP.EVAPS3.OP_Stop.OK,
	I_STOP_IAD_OK := TRUE,
	I_POMPAGE_SEC_OK := NOT PRG_POMPAGE.POMPAGE.OP_Pompage_Sec.AR,
	I_TH_ATM := PRG_POMPAGE.POMPAGE.TH_Atm,
	I_DOOR := PRG_POMPAGE.DOOR,
	I_STOP_CONTROLLER_OK := PRG_EVAP.XTC3.STATE_STOP,// OR PRG_EVAP.XTC3.STATE_NOK,
	I_STOP_EFFLUVAGE_OK := TRUE,
	I_STOP_GAZ_OK := PRG_GAZ.LIGNE_GAZ[1].OP_ARRET.OK AND PRG_GAZ.LIGNE_GAZ[2].OP_ARRET.OK AND PRG_GAZ.LIGNE_GAZ[3].OP_ARRET.OK AND PRG_GAZ.LIGNE_GAZ[4].OP_ARRET.OK
					   AND PRG_GAZ.REGULATION_GAZ_L1.OP_ARRET.OK AND PRG_GAZ.REGULATION_GAZ_L2.OP_ARRET.OK ,
	I_STOP_CHAUFFAGE_OK := TRUE,
	I_STOP_MVTS_OK := PRG_MOUVEMENT_PS.ROTATION_PS.OP_Arret.OK,
	I_INIT_POSE_OK := TRUE,
	I_INIT_PRISE_OK := TRUE,
	I_PURGE_EC	:= FALSE,
	CO_Inter:= MACHINE.RQ_Inter_Prod,
	CO_Stop_Prod:= MACHINE.RQ_Stop_Prod OR EXECPROC.RQ_EXEC_STEP[15],
	CO_Init_Prod:= MACHINE.RQ_Prep_Prod,
	CO_init:= MACHINE.RQ_Init,
	STATE_OK=> );	

(*étape de pompage *)
EXECPROC.EN_EXEC_STEP[1] 		:= 	PRG_POMPAGE.POMPAGE.OP_Pompage_Sec.AUTOR_PLC;
EXECPROC.I_EXEC_STEP_OK[1] 		:= 	PRG_POMPAGE.O_STEP_PUMPING_OK;
EXECPROC.EN_NEXT_STEP[1] 		:= 	PRG_POMPAGE.POMPAGE.OP_Pompage_sec.OK;
(*etape d'isolement*)
EXECPROC.EN_EXEC_STEP[2] 		:= 	PRG_POMPAGE.POMPAGE.OP_Isolement.AUTOR_PLC;
EXECPROC.I_EXEC_STEP_OK[2]		:=	PRG_POMPAGE.POMPAGE.OP_Isolement.OK;
EXECPROC.EN_NEXT_STEP[2] 		:= 	FALSE;
(*etape de marche pompes*)
EXECPROC.EN_EXEC_STEP[3] 		:= 	PRG_POMPAGE.POMPAGE.OP_Marche_Pompes.AUTOR_PLC;
EXECPROC.I_EXEC_STEP_OK[3]		:=	PRG_POMPAGE.POMPAGE.OP_Marche_Pompes.OK;
EXECPROC.EN_NEXT_STEP[3] 		:= 	TRUE;
(*Etape d'arrêt des pompes*)
EXECPROC.EN_EXEC_STEP[4] 		:= 	PRG_POMPAGE.POMPAGE.OP_Arret_Pompes.AUTOR_PLC;
EXECPROC.I_EXEC_STEP_OK[4]		:=	PRG_POMPAGE.POMPAGE.OP_Arret_Pompes.OK;
EXECPROC.EN_NEXT_STEP[4] 		:= 	TRUE;
(*Etape de regeneration*)
EXECPROC.EN_EXEC_STEP[5] 		:= 	PRG_POMPAGE.POMPAGE.OP_Regen.AUTOR_PLC;
EXECPROC.I_EXEC_STEP_OK[5]		:=	PRG_POMPAGE.POMPAGE.OP_Regen.OK;
EXECPROC.EN_NEXT_STEP[5] 		:= 	TRUE;
(*Etape de ventilation*)
EXECPROC.EN_EXEC_STEP[6] 		:= 	PRG_POMPAGE.POMPAGE.OP_Ventilation.AUTOR_PLC;
EXECPROC.I_EXEC_STEP_OK[6]		:=	PRG_POMPAGE.POMPAGE.OP_Ventilation.OK;
EXECPROC.EN_NEXT_STEP[6] 		:= 	TRUE;
(*Point d'arrêt*)
EXECPROC.EN_EXEC_STEP[7]		:=	TRUE;
EXECPROC.I_EXEC_STEP_OK[7]		:=	STEP_USER_ACK.STATE_OK;
EXECPROC.EN_NEXT_STEP[7] 		:= 	FALSE;
(*Etape empilement-evaporation*)
EXECPROC.EN_EXEC_STEP[8]		:= 	(PRG_POMPAGE.POMPAGE.OP_Pompage_Sec.OK OR PRG_POMPAGE.POMPAGE.OP_Pompage_Proc.OK)
							    	AND (NOT PRG_EVAP.QZ1.DEF_QZ.DEF OR MODE_QUARTZ_PROD.STATE_Mode);
EXECPROC.I_EXEC_STEP_OK[8]		:=	STEP_EMPILEMENT.STATE_OK;
EXECPROC.EN_NEXT_STEP[8] 		:= 	FALSE;
EXECPROC.PRM_NEXT_STEP_EXT[8]	:=	FALSE;
(*synchro horaire*)
EXECPROC.EN_EXEC_STEP[9]		:=	TRUE;
EXECPROC.I_EXEC_STEP_OK[9]		:=	STEP_SYNHRO_HORAIRE.STATE_OK ;
EXECPROC.EN_NEXT_STEP[9] 		:= 	TRUE;
EXECPROC.PRM_NEXT_STEP_EXT[9]	:=	FALSE;
(*timer*)
EXECPROC.EN_EXEC_STEP[10]		:=	TRUE;
EXECPROC.I_EXEC_STEP_OK[10]		:=	STEP_TIMER.STATE_OK ;
EXECPROC.EN_NEXT_STEP[10] 		:= 	TRUE;
EXECPROC.PRM_NEXT_STEP_EXT[10]	:=	FALSE;
(*rotation PS*)
EXECPROC.EN_EXEC_STEP[11]		:=	PRG_MOUVEMENT_PS.ROTATION_PS.OP_Rotation.AUTOR_PLC ;
EXECPROC.I_EXEC_STEP_OK[11]		:=	PRG_MOUVEMENT_PS.ROTATION_PS.OP_Rotation.OK ;
EXECPROC.EN_NEXT_STEP[11] 		:= 	FALSE;
EXECPROC.PRM_NEXT_STEP_EXT[11]	:=	FALSE;
(*arret rotation PS*)
EXECPROC.EN_EXEC_STEP[12]		:=	PRG_MOUVEMENT_PS.ROTATION_PS.OP_ARRET.AUTOR_PLC ;
EXECPROC.I_EXEC_STEP_OK[12]		:=	PRG_MOUVEMENT_PS.ROTATION_PS.OP_ARRET.OK ;
EXECPROC.EN_NEXT_STEP[12] 		:= 	FALSE;
EXECPROC.PRM_NEXT_STEP_EXT[12]	:=	FALSE;
(*Etape effluvage*)
EXECPROC.EN_EXEC_STEP[13]		:=	FALSE ;
EXECPROC.I_EXEC_STEP_OK[13]		:=	STEP_EFFLUVAGE.STATE_OK  ;
EXECPROC.EN_NEXT_STEP[13] 		:= 	STEP_EFFLUVAGE.AUTOR_NEXT_STEP;
EXECPROC.PRM_NEXT_STEP_EXT[13]	:=	TRUE;
(*test de remontée de pression*)
EXECPROC.EN_EXEC_STEP[14]		:= 	PRG_POMPAGE.POMPAGE.OP_Pompage_Sec.OK ;
EXECPROC.I_EXEC_STEP_OK[14]		:=	PRG_POMPAGE.POMPAGE.OP_Test_RP.OK  ;
EXECPROC.EN_NEXT_STEP[14] 		:= 	FALSE;
EXECPROC.PRM_NEXT_STEP_EXT[14]	:=	FALSE;
(*arret procédé*)
EXECPROC.EN_EXEC_STEP[15]		:=	TRUE;
EXECPROC.I_EXEC_STEP_OK[15]		:=	INIT_MACHINE.STATE_OK  ;
EXECPROC.EN_NEXT_STEP[15] 		:= 	FALSE;
EXECPROC.PRM_NEXT_STEP_EXT[15]	:=	FALSE;
(*boucle saut*)
EXECPROC.EN_EXEC_STEP[16]		:=	STEP_BOUCLE.AUTOR_STEP;
EXECPROC.I_EXEC_STEP_OK[16]		:=	STEP_BOUCLE.STATE_OK;
EXECPROC.EN_NEXT_STEP[16] 		:= 	FALSE;
EXECPROC.PRM_NEXT_STEP_EXT[16]	:=	FALSE;
(*Lancement mode eco*)
EXECPROC.EN_EXEC_STEP[17]		:=	TRUE;
EXECPROC.I_EXEC_STEP_OK[17]		:=	MACHINE.I_Standby_Ok;
EXECPROC.EN_NEXT_STEP[17] 		:= 	FALSE;
EXECPROC.PRM_NEXT_STEP_EXT[17]	:=	FALSE;
(*Arrêt mode eco*)
EXECPROC.EN_EXEC_STEP[18]		:=	TRUE;
EXECPROC.I_EXEC_STEP_OK[18]		:=	NOT MACHINE.I_Standby_Ok AND MACHINE.I_WakeUp_Ok;
EXECPROC.EN_NEXT_STEP[18] 		:= 	FALSE;
EXECPROC.PRM_NEXT_STEP_EXT[18]	:=	FALSE;
(*Régénération partielle*)
EXECPROC.EN_EXEC_STEP[19] 		:= 	PRG_POMPAGE.POMPAGE.OP_Regen_Part.AUTOR_PLC;
EXECPROC.I_EXEC_STEP_OK[19]		:=	PRG_POMPAGE.POMPAGE.OP_Regen_Part.OK;
EXECPROC.EN_NEXT_STEP[19] 		:= 	TRUE;

IF MACHINE.RQ_Start_Proc_WeekEnd THEN (*Assignation du procédé week-end*)
	EXECPROC.PRM_PROCESS_NAME :=  MACHINE.PRM_PROCESS_NAME_WEEKEND;
	EXECPROC.PRM_PROCESS :=  MACHINE.PRM_PROCESS_WEEKEND;
	EXECPROC.PRM_BATCH := MACHINE.PRM_BATCH_WEEKEND;
	EXECPROC.PRM_RECORD :=  MACHINE.PRM_RECORD_WEEKEND;
END_IF

EXECPROC(
	I_ON:= 					MACHINE.RQ_Start_Prod OR MACHINE.RQ_Start_Proc_WeekEnd,
	I_INTER_PROC:= 			MACHINE.STATE_Inter_Prod,
	PRM_NEXT_STEP:=			STEP_BOUCLE.O_NEXT_STEP,
	PRM_BOUCLE:=			STEP_BOUCLE.RQ_BOUCLE,
	PRM_SAUT:=				STEP_BOUCLE.RQ_SAUT,
	RQ_EXEC_STEP=>);
	
	
(*Gestion quartz en production*)
MODE_QUARTZ_PROD.I_QF[1]	:=	PRG_EVAP.QZ1.STATE_QF1;
MODE_QUARTZ_PROD.I_QF[2]	:=	PRG_EVAP.QZ1.STATE_QF2;
MODE_QUARTZ_PROD.I_QF[3]	:=	PRG_EVAP.QZ1.STATE_QF3;
MODE_QUARTZ_PROD.I_QF[4]	:=	PRG_EVAP.QZ1.STATE_QF4;
MODE_QUARTZ_PROD.I_QF[5]	:=	PRG_EVAP.QZ1.STATE_QF5;
MODE_QUARTZ_PROD.I_QF[6]	:=	PRG_EVAP.QZ1.STATE_QF6;
MODE_QUARTZ_PROD(
	I_Prod:=				MACHINE.STATE_Prod,
	I_Evap:=				STEP_EMPILEMENT.STATE_EVAP,
	I_CD6T:=				PRG_EVAP.XTC3.IN_CD36T,
	I_Current_Quartz:=		PRG_EVAP.QZ1.STATE_POSITION,	
	);
	

(*gestion de la sauvegarde des paramètres persistents : on fait retomber l'état param_system_ok*)
IF RQ_PARAM_SYSTEM THEN
 	PARAM_SYSTEM_OK	 := FALSE;
END_IF

(*DEBUGECO*)
IF EXECPROC.RQ_EXEC_STEP[17] THEN
	VAR_Mem_Eco	:=	TRUE;
ELSIF NOT EXECPROC.I_ON THEN
	VAR_Mem_Eco	:=	FALSE;
END_IF

(*Appel des programmes*)
PRG_POMPAGE();
PRG_User();
PRG_SERVITUDES();
PRG_MOUVEMENT_PS();
PRG_EFFLUVAGE();
PRG_GAZ();
PRG_EVAP();
PRG_SEC();
PRG_DEF_MANAGEMENT();
PRG_VERRINE();
PRG_INFO_CLIENT();

IF NOT PARAM_SYSTEM_OK THEN
	RQ_PARAM_SYSTEM			:=	FALSE;
	PARAM_SYSTEM_OK			:=	TRUE;
	RQ_SAV_PERSISTENT		:=	TRUE;
END_IF;

(*Gestion du passage en mode manu non securisé*)
(*enclenchement timer sur appui prolongé sur bouton*)
TIMER_SECU_OFF.PT 	:= 	T#5s;
TIMER_SECU_OFF.IN 		:= 	IHM_SHUNT_SECU;
TIMER_SECU_OFF();
(*gestion de la variable globale *)
IF TIMER_SECU_OFF.Q THEN
	MANUAL_SAFETY_OFF 	:= 	TRUE;
ELSIF IHM_SECU_ON THEN (*reprise sur appui simple sur bouton*)
	MANUAL_SAFETY_OFF 	:= 	FALSE;
	IHM_SECU_ON			:= 	FALSE;
END_IF
(*gestion de la progress bar : utilité du *123.???*)
STATE_PROGRESS_BAR_MANU :=  REAL_TO_USINT((TIME_TO_REAL(TIMER_SECU_OFF.ET)/TIME_TO_REAL(TIMER_SECU_OFF.PT)) * 123);

(*GESTION TRAC*)
(*reset demande enregistrement manuel*)
IF MACHINE.RQ_Prep_Prod OR MACHINE.RQ_Stop_Prod THEN
	Enr_TRAC	:=	FALSE;
END_IF
(*demande enregistrement TRAC*)
TRAC_RECORD	:=	Enr_TRAC OR (EXECPROC.PRM_RECORD AND MACHINE.STATE_Prod AND NOT MACHINE.STATE_Pause_TrAC); 
(*nom enregistrement*)
IF MACHINE.STATE_Prod THEN
	TRAC_PROCESS_NAME	:=	EXECPROC.PRM_PROCESS_NAME;
ELSE
	TRAC_PROCESS_NAME	:=	'Standby';
END_IF
(*export en fin production*)
TRAC_EXPORT_AUTO:= MACHINE.STATE_Prod AND NOT MACHINE.STATE_Pause_TrAC AND EXECPROC.PRM_RECORD;
(*enregistrement lent sur éco-veille*)
TRAC_SLOW_RECORD:=PRG_EVAP.ECO_MODE;



(*Bit de clignotement*)
BIT_1s(PRM_PERIOD:= T#1s );

(*Etape d'acquittement opérateur*)
STEP_USER_ACK(I_ON:=EXECPROC.RQ_EXEC_STEP[7]
						(*OR EXECPROC.RQ_EXEC_STEP[24]*));

(*Etapes synchro / tempo*)
STEP_SYNHRO_HORAIRE(I_ON:=EXECPROC.RQ_EXEC_STEP[9]);
STEP_TIMER(	I_ON:=						EXECPROC.RQ_EXEC_STEP[10],
			I_ROTATION_OK:= 			PRG_MOUVEMENT_PS.ROTATION_PS.OP_Rotation.OK,
			I_STOP_ROT_PS_OK:= 			PRG_MOUVEMENT_PS.ROTATION_PS.OP_ARRET.OK,
			I_NO_ROTATION_PS:= 			PRG_MOUVEMENT_PS.PRM_Vitesse = 0,		(*Pas de rotation PS si consigne nulle*)
);
(*Etape boucle/saut*)
(*marche sur exécution étape*)
IF EXECPROC.RQ_EXEC_STEP[16] THEN
	STEP_BOUCLE.I_ON	:=	TRUE;
(*arrêt sur lecture etape suivante (2), interruption procédé (8), procédé à l'arrêt (0)*)
ELSIF EXECPROC.OP_RUN.Etape.2 OR EXECPROC.OP_RUN.Etape.8 OR EXECPROC.OP_RUN.Etape.0 THEN
	STEP_BOUCLE.I_ON	:=	FALSE;
END_IF
STEP_BOUCLE(
	RESET:= 				NOT MACHINE.STATE_Prod,
	I_CURRENT_STEP:= 		EXECPROC.STATE_STEP,
	 );

(*Etape d'effluvage*)
//STEP_EFFLUVAGE(
//	I_ON:= 						EXECPROC.RQ_EXEC_STEP[13],
//	I_POMPAGE_SEC_OK:= 			PRG_POMPAGE.POMPAGE.OP_Pompage_Sec.OK,
//	I_POMPAGE_PRIM_OK:=			PRG_POMPAGE.POMPAGE.OP_Pompage_Prim.OK,
//	I_ROTATION_OK:= 			PRG_MOUVEMENT_PS.ROTATION_PS.OP_Rotation.OK,
//	I_STOP_ROT_PS_OK:= 			PRG_MOUVEMENT_PS.ROTATION_PS.OP_ARRET.OK,
//	I_NO_ROTATION_PS:= 			PRG_MOUVEMENT_PS.ROTATION_PS.PRM_Vitesse = 0,		(*Pas de rotation PS si consigne nulle*)
//	I_ISOLEMENT_OK:=			PRG_POMPAGE.POMPAGE.OP_Isolement.OK,
//	I_MARCHE_GAZ1_OK:= 			PRG_GAZ.LIGNE_GAZ[3].OP_MARCHE.OK,
//	I_ARRET_GAZ1_OK:= 			PRG_GAZ.LIGNE_GAZ[3].OP_ARRET.OK,
//	I_MARCHE_GAZ2_OK:=			PRG_GAZ.LIGNE_GAZ[4].OP_MARCHE.OK,
//	I_ARRET_GAZ2_OK:=			PRG_GAZ.LIGNE_GAZ[4].OP_ARRET.OK,
//	M_NEXT_STEP:=				EXECPROC.RQ_NEXT_STEP,
//	I_MARCHE_EFFLUVAGE_OK:=		FALSE,(*PRG_EFFLUVAGE.Effluvage.OP_Marche_Eff.OK,*)
//	I_ARRET_EFFLUVAGE_OK:= 		TRUE,(*PRG_EFFLUVAGE.Effluvage.OP_Arret_Eff.OK,*)
//	TH_EFFLUVAGE:=				PRG_POMPAGE.M11.STATE_Seuil[12],				(*Pression de vide avant effluvage*)
//	TH_PPRIM_AUTOR:= 			NOT(PRG_POMPAGE.M11.STATE_Seuil[3]),			(*Pression d'autorisation de pompage primaire*)
//	I_MODE_REPRISE:= 			EXECPROC.STATE_reprise,
//	PRM_PR_EFFLUVAGE:=  ,
//	PRM_TEMPS_EFF:= ,
//	CONS_TPS_EFFLUVAGE:=		T#0MS,(*PRG_EFFLUVAGE.Effluvage.PRM_TPS_effluvage,*)
//	RQ_POMPAGE_PRIM=> ,
//	RQ_ISOLEMENT=> ,
//	RQ_MARCHE_EFFLUVAGE=> ,
//	RQ_ARRET_EFFLUVAGE=> ,
//	RQ_ROTATION_PS=> ,
//	STATE_OK=> ,
//	STATUS=> ,
//	CONS_FLOW_GAZ_1 := 				PRG_GAZ.LIGNE_GAZ[3].PRM_Flow,
//	CONS_FLOW_GAZ_2 := 				PRG_GAZ.LIGNE_GAZ[4].PRM_Flow,);

(*Etape d'empilement*)
STEP_EMPILEMENT(
	I_ON:= 							EXECPROC.RQ_EXEC_STEP[8],
	I_MODE_REPRISE:= 				EXECPROC.STATE_reprise,
	I_ROTATION_PS_OK:= 				PRG_MOUVEMENT_PS.ROTATION_PS.OP_Rotation.OK,
	I_TILT_PS_OK:=					TRUE,														(*Pas de tilt*)
	I_STOP_ROT_PS_OK:= 				PRG_MOUVEMENT_PS.ROTATION_PS.OP_ARRET.OK,
	I_STOP_TILT_PS_OK:=				TRUE,														(*Pas de tilt*)
	I_NO_ROTATION_PS:=				(PRG_MOUVEMENT_PS.PRM_Vitesse = 0),							(*Pas de rotation PS si consigne nulle*)
	I_MODE_TILT:=					1,															(*Pas de tilt*)
	I_ACTION_CONTROLEUR_OK:=		PRG_EVAP.XTC3.STATE_ACTION_OK,
	I_CONTROLEUR_PHASE:= 			PRG_EVAP.XTC3.STATE_Phase,
	I_CONTROLEUR_STOPPED:= 			PRG_EVAP.XTC3.STATE_STOP,
	I_PROG_CONTROLEUR_OK:= 			PRG_EVAP.XTC3.STATE_Prog_Layer_OK,
	I_END_DEPOT:= 					PRG_EVAP.XTC3.OUT_END_OF_PROCESS OR PRG_EVAP.EVAPS1.STATE_END_DEPOT_PFIXE
									OR PRG_EVAP.EVAPS2.STATE_END_DEPOT_PFIXE OR PRG_EVAP.EVAPS3.STATE_END_DEPOT_PFIXE,
	I_Global_Thick := 				PRG_EVAP.XTC3.STATE_Thickness,
	I_Global_Rate := 				PRG_EVAP.XTC3.STATE_Rate,
	I_N_SEGMENT_S1 := 				PRG_EVAP.EVAPS1.STATE_Segment,
	I_N_SEGMENT_S2 := 				PRG_EVAP.EVAPS2.STATE_Segment,
	I_N_SEGMENT_S3 :=				PRG_EVAP.EVAPS3.STATE_Segment,
	I_MARCHE_CHAUFFAGE_OK:= 		TRUE,		(*Pas de chauffage*)
	I_ARRET_CHAUFFAGE_OK:= 			TRUE,		(*Pas de chauffage*)
	I_ARRET_GAZ1_OK:= 				PRG_GAZ.LIGNE_GAZ[1].OP_ARRET.OK,
	I_ARRET_GAZ2_OK:=				PRG_GAZ.LIGNE_GAZ[2].OP_ARRET.OK,
	I_MARCHE_POMPAGE_SEC_OK :=		PRG_POMPAGE.POMPAGE.OP_Pompage_Sec.OK,
	I_MARCHE_POMPAGE_PROC_OK :=		PRG_POMPAGE.POMPAGE.OP_Pompage_Proc.OK,
	I_MARCHE_IAD_OK:= 				TRUE,				(*Pas d'IAD*)
	I_ARRET_IAD_OK:= 				TRUE,				(*Pas d'IAD*)
	I_MARCHE_GAZ1_OK:= 				PRG_GAZ.LIGNE_GAZ[1].OP_MARCHE.OK,
	I_MARCHE_GAZ2_OK:= 				PRG_GAZ.LIGNE_GAZ[2].OP_MARCHE.OK,
	I_NO_MORE_LAYER_ANT:= 			TRUE,			(*Pas de gestion de couche anticipée dans ACSoft*)
	I_LAYER_ANT_LOADING_OK:= 		TRUE,			(*Pas de gestion de couche anticipée dans ACSoft*)
	I_PREP_SOURCE1_OK:=				PRG_EVAP.EVAPS1.STATE_PREP_OK ,
	I_PREP_SOURCE2_OK:= 			PRG_EVAP.EVAPS2.STATE_PREP_OK ,
	I_PREP_SOURCE3_OK:=				PRG_EVAP.EVAPS3.STATE_PREP_OK ,
	I_CLOT_SOURCE1_OK:= 			PRG_EVAP.EVAPS1.STATE_CLOT_OK ,
	I_CLOT_SOURCE2_OK:= 			PRG_EVAP.EVAPS2.STATE_CLOT_OK ,
	I_CLOT_SOURCE3_OK:= 			PRG_EVAP.EVAPS3.STATE_CLOT_OK ,
	I_STAB_CHAUFFAGE_OK:=			TRUE,			(*Pas de chauffage*)
	PRM_TPS_PREPA_SOURCE1:= 		PRG_EVAP.EVAPS1.STATE_TEMPS_PREPARATION,
	PRM_TPS_PREPA_SOURCE2:= 		PRG_EVAP.EVAPS2.STATE_TEMPS_PREPARATION,
	PRM_TPS_PREPA_SOURCE3:= 		PRG_EVAP.EVAPS3.STATE_TEMPS_PREPARATION,
	PRM_SOURCE1_RATE:=				PRG_EVAP.EVAPS1.PRM_Rate,
	PRM_SOURCE2_RATE:= 				PRG_EVAP.EVAPS2.PRM_Rate,
	PRM_SOURCE3_RATE:= 				PRG_EVAP.EVAPS3.PRM_Rate,
	I_SOURCE1_ARRET:= 				PRG_EVAP.EVAPS1.OP_Marche.Etape.0 OR PRG_EVAP.EVAPS1.OP_Marche.Etape.16,
	I_SOURCE2_ARRET:= 				PRG_EVAP.EVAPS2.OP_Marche.Etape.0 OR PRG_EVAP.EVAPS2.OP_Marche.Etape.16,
	I_SOURCE3_ARRET:= 				PRG_EVAP.EVAPS3.OP_Marche.Etape.0 OR PRG_EVAP.EVAPS3.OP_Marche.Etape.16,
	I_EVAP1_OK:=					PRG_EVAP.EVAPS1.STATE_EVAP,
	I_EVAP2_OK:=					PRG_EVAP.EVAPS2.STATE_EVAP,
	I_EVAP3_OK:=					PRG_EVAP.EVAPS3.STATE_EVAP,
	I_STOP_EVAP1_OK:= 				PRG_EVAP.EVAPS1.STATE_AR,
	I_STOP_EVAP2_OK:= 				PRG_EVAP.EVAPS2.STATE_AR,
	I_STOP_EVAP3_OK:= 				PRG_EVAP.EVAPS3.STATE_AR,
	I_STOP_EVAP4_OK:=  				TRUE,
	I_DOME_IN_POSITION:= 			TRUE,
	I_SOURCE1_PREFU:=				PRG_EVAP.EVAPS1.STATE_PREFU,
	I_SOURCE2_PREFU:= 				PRG_EVAP.EVAPS2.STATE_PREFU,
	I_SOURCE3_PREFU:= 				PRG_EVAP.EVAPS3.STATE_PREFU,
	I_SOURCE1_IDLE:= 				PRG_EVAP.EVAPS1.STATE_IDLE,
	I_SOURCE2_IDLE:= 				PRG_EVAP.EVAPS2.STATE_IDLE,
	I_SOURCE3_IDLE:= 				PRG_EVAP.EVAPS3.STATE_IDLE,
	CONS_FLOW_GAZ_1 := 				PRG_GAZ.LIGNE_GAZ[1].PRM_Flow,
	CONS_FLOW_GAZ_2 := 				PRG_GAZ.LIGNE_GAZ[2].PRM_Flow,
);

STEP_EMPILEMENT.I_ARRET_REGUL_GAZ_OK[1]:= PRG_GAZ.REGULATION_GAZ_L1.OP_ARRET.OK;
STEP_EMPILEMENT.I_ARRET_REGUL_GAZ_OK[2]:= PRG_GAZ.REGULATION_GAZ_L2.OP_ARRET.OK;

IF (STEP_EMPILEMENT.CONS_MODE = 0 OR STEP_EMPILEMENT.CONS_MODE = 1) AND STEP_EMPILEMENT.RQ_MARCHE_POMPAGE_PROC THEN
	PRG_POMPAGE.POMPAGE.VS11.PRM_Mode			:=	USINT_TO_BOOL( STEP_EMPILEMENT.CONS_MODE);
	PRG_POMPAGE.POMPAGE.VS11.PRM_Pression		:= 	STEP_EMPILEMENT.CONS_PRESSURE;
	PRG_POMPAGE.POMPAGE.VS11.PRM_Position		:= 	STEP_EMPILEMENT.CONS_POSITION;
	PRG_POMPAGE.POMPAGE.VS11.PRM_W_Pr_HI		:= 	STEP_EMPILEMENT.CONS_HI_PRESSURE;
	PRG_POMPAGE.POMPAGE.VS11.PRM_W_Pr_LO		:= 	STEP_EMPILEMENT.CONS_LOW_PRESSURE;
	PRG_POMPAGE.POMPAGE.VS11.PRM_Tim_W_Pr		:= 	STEP_EMPILEMENT.CONS_TIM_PRESSURE;
END_IF

IF STEP_EMPILEMENT.CONS_MODE = 2 AND STEP_EMPILEMENT.RQ_MARCHE_REGUL_GAZ[1] THEN
	PRG_GAZ.REGULATION_GAZ_L1.PRM_Pressure		:= 	STEP_EMPILEMENT.CONS_PRESSURE;
	PRG_GAZ.REGULATION_GAZ_L1.PRM_Pos_Vanne		:= 	STEP_EMPILEMENT.CONS_POSITION;
	PRG_GAZ.REGULATION_GAZ_L1.PRM_Pressure_H	:= 	STEP_EMPILEMENT.CONS_HI_PRESSURE;
	PRG_GAZ.REGULATION_GAZ_L1.PRM_Pressure_L	:= 	STEP_EMPILEMENT.CONS_LOW_PRESSURE;
	PRG_GAZ.REGULATION_GAZ_L1.PRM_Tim_Stab		:= 	STEP_EMPILEMENT.CONS_TIM_PRESSURE;
END_IF

IF STEP_EMPILEMENT.CONS_MODE = 3 AND STEP_EMPILEMENT.RQ_MARCHE_REGUL_GAZ[2] THEN
	PRG_GAZ.REGULATION_GAZ_L2.PRM_Pressure		:= 	STEP_EMPILEMENT.CONS_PRESSURE;
	PRG_GAZ.REGULATION_GAZ_L2.PRM_Pos_Vanne		:= 	STEP_EMPILEMENT.CONS_POSITION;
	PRG_GAZ.REGULATION_GAZ_L2.PRM_Pressure_H	:= 	STEP_EMPILEMENT.CONS_HI_PRESSURE;
	PRG_GAZ.REGULATION_GAZ_L2.PRM_Pressure_L	:= 	STEP_EMPILEMENT.CONS_LOW_PRESSURE;
	PRG_GAZ.REGULATION_GAZ_L2.PRM_Tim_Stab		:= 	STEP_EMPILEMENT.CONS_TIM_PRESSURE;
END_IF


VAR_FB_WritePersistentData(
	NETID:=		'' ,
	PORT:= 		801,
	START:=		RQ_SAV_PERSISTENT (*OR  VAR_Compteur.VAR_Cpt_Temps.TIMER_Valid_On.Q, *) , (*ajout sauvegarde périodique toutes les heures*)
	TMOUT:= 	T#2s000ms,
	MODE:= 		SPDM_VAR_BOOST,	(*ecriture en plusieur cycle automate*)
	BUSY=>		FM_BUSY.CLK ,
	ERR=> 		FM_ERROR.CLK,
	ERRID=> );
FM_BUSY();
FM_ERROR();


IF RQ_SAV_PERSISTENT AND (FM_BUSY.Q OR FM_ERROR.Q)  THEN
	RQ_SAV_PERSISTENT	:=	FALSE;
END_IF;


(*Divers*)
CPT_USURE.I_Machine_prod		:=	MACHINE.STATE_Prod;
CPT_USURE.I_PRE_EVAP_ON			:=	STEP_EMPILEMENT.I_SOURCE1_PREFU;
CPT_USURE.I_EVAP_OFF			:=	STEP_EMPILEMENT.I_SOURCE1_IDLE;
CPT_USURE.I_EVAP_ON				:=	PRG_EVAP.EVAPS1.STATE_EVAP AND PRG_EVAP.CC11.STATE_On;
CPT_USURE.I_LAYER_LOAD_OK		:=	STEP_EMPILEMENT.OP_RUN.Etape.6;

CPT_USURE();

(*Lancement du .exe de démarrage de process*)
Process.PATHSTR	:= 	'C:\Machine\Verif_AC_Soft\Verif_Ac_Soft.exe';
(*process.PATHSTR:= 'C:\windows\notepad.exe';*)
Process.DIRNAME	:= 	'C:\Machine\Verif_AC_Soft';
Process.START	:= 	bStartVerif;
Process();

(*gestion inactivité*)
TIMER_Inactivite.IN	:= 	MACHINE.STATE_Auto
						AND NOT MACHINE.STATE_Prod
						AND MACHINE.CONF_Standby_Auto
						AND PRG_EFFLUVAGE.STATE_Ar
						AND PRG_EVAP.STATE_Ar
						AND PRG_GAZ.STATE_Ar
						AND PRG_MOUVEMENT_PS.STATE_Ar;
TIMER_Inactivite.PT	:=	MACHINE.CONF_Tps_Inactivite;
TIMER_Inactivite();

END_PROGRAM

// ---- POUs/FONCTION DE BASE/BLOCK_CLIGNOTANT.TcPOU
FUNCTION_BLOCK BLOCK_CLIGNOTANT
VAR_INPUT
	PRM_PERIOD:	TIME;
END_VAR
VAR_OUTPUT
	STATE: 		BOOL;
END_VAR
VAR
	TIMER_ON:	TP;
	TIMER_OFF:	TP;
END_VAR

TIMER_ON(IN:=NOT TIMER_OFF.Q ,PT:= PRM_PERIOD);
TIMER_OFF(IN:=NOT TIMER_ON.Q,PT:=PRM_PERIOD);
STATE := TIMER_ON.Q;

END_FUNCTION_BLOCK

// ---- POUs/Fonction/FONCTION MODEMARCHE/BLOCK_USER_ACK.TcPOU
FUNCTION_BLOCK BLOCK_USER_ACK
VAR_INPUT
	PRM_TEXT:		STRING(255);
	I_ON:			BOOL;
	M_GOON:		BOOL;
END_VAR
VAR_OUTPUT
	STATE_EC:	BOOL;
	STATE_OK:		BOOL;
END_VAR
VAR
END_VAR

IF  I_ON AND NOT STATE_OK THEN
	STATE_EC := TRUE;
END_IF;
IF NOT I_ON OR STATE_OK THEN
	STATE_EC:=FALSE;
END_IF

IF I_ON AND M_GOON THEN
	STATE_OK:=TRUE;
ELSIF NOT I_ON THEN
	STATE_OK:=FALSE;
END_IF

END_FUNCTION_BLOCK

// ---- POUs/Fonction/FONCTION MODEMARCHE/BLOCK_SYNCHRO_HORAIRE.TcPOU
FUNCTION_BLOCK BLOCK_SYNCHRO_HORAIRE
VAR_INPUT
	I_ON:		BOOL;
	PRM_DAY:	USINT;
	PRM_HOUR:	USINT;
	PRM_MINUTE: USINT;
END_VAR
VAR_OUTPUT
	STATE_OK:	BOOL;
END_VAR
VAR

END_VAR

(*etat ok*)
STATE_OK := I_ON AND
			((PRM_DAY = PRG_SEC.STATE_DT.wDayOfWeek) OR (PRM_DAY = 7)) AND
			(PRM_HOUR = PRG_SEC.STATE_DT.whour) AND
			(PRM_MINUTE = PRG_SEC.STATE_DT.wMinute);

END_FUNCTION_BLOCK

// ---- POUs/Programme/PRG_SEC.TcPOU
PROGRAM PRG_SEC
VAR
(***********************************************************************************)
(*Fonction de récupération de l'heure locale (Windows) par simple mise à 1 du bEnable au démarrage*)
(* Version 0 - GV - 06/2017 - Affaire 10315    *)
(***********************************************************************************)

	fbTime : FB_LocalSystemTime := ( bEnable := TRUE, dwCycle := 1);


	_ms:			UINT;
	_date:			DT;
	m_string:			STRING;
	STATE_Date:	STRING;
	STATE_Time:	STRING;
	STATE_DT:		TIMESTRUCT;

	STATE_Time_OK:	BOOL;

	VERROU : 		BOOL:=FALSE;
END_VAR

fbTime();

_Date	:=	SYSTEMTIME_TO_DT(fbTime.systemTime);
_ms		:=	WORD_TO_UINT(fbTime.systemTime.wMilliseconds);

m_string			:= 	CONCAT(	WORD_TO_STRING(fbTime.systemTime.wDay),'/');
IF fbTime.systemTime.wMonth < 16#000A THEN		(*mois < 10*)
	m_string 		:=	CONCAT(	m_string,'0');
	m_string 		:=	CONCAT(	m_string,WORD_TO_STRING(fbTime.systemTime.wMonth) );
ELSE
	m_string 		:=	CONCAT(	m_string,WORD_TO_STRING(fbTime.systemTime.wMonth) );
END_IF;
m_string			:=	CONCAT(	m_string ,'/' );
m_string			:=	CONCAT(	m_string , WORD_TO_STRING(fbTime.systemTime.wYear) );
STATE_DATE 		:= 	m_string;

m_string 			:= 	CONCAT(	WORD_TO_STRING(fbTime.systemTime.wHour),':');
IF fbTime.systemTime.wMinute < 16#000A THEN
	m_string 		:=	CONCAT(	m_string,'0');
	m_string 		:=	CONCAT(	m_string,WORD_TO_STRING(fbTime.systemTime.wMinute) );
ELSE
	m_string 		:=	CONCAT(	m_string,WORD_TO_STRING(fbTime.systemTime.wMinute) );
END_IF;
m_string 			:=	CONCAT(	m_string,':');
IF fbTime.systemTime.wSecond < 16#000A THEN
	m_string 		:=	CONCAT(	m_string,'0');
	m_string 		:=	CONCAT(	m_string,WORD_TO_STRING(fbTime.systemTime.wSecond) );
ELSE
	m_string 		:=	CONCAT(	m_string,WORD_TO_STRING(fbTime.systemTime.wSecond) );
END_IF;
STATE_Time 		:= 	m_string;
STATE_DT	 	:= 	fbTime.systemTime;

STATE_Time_Ok	:=	(fbTime.systemTime.wYear <> 0);

END_PROGRAM

// ---- POUs/Fonction/FONCTION MODEMARCHE/BLOCK_STEP_TIMER.TcPOU
FUNCTION_BLOCK BLOCK_STEP_TIMER
VAR_INPUT
	I_ON:					BOOL;
	PRM_TIME:				DINT;
	OP_RUN:					BLOCK_G7;				(*Grafcet de gestion de l'étape timer*)
	I_ROTATION_OK:			BOOL;					(*Condition rotation ok*)
	I_STOP_ROT_PS_OK:		BOOL;					(*Retour rotation PS à l'arrêt*)
	I_NO_ROTATION_PS:		BOOL;					(*Pas de rotation PS si consigne nulle*)
END_VAR
VAR_OUTPUT
	RQ_ROTATION_PS:			BOOL;
	RQ_STOP_ROTATION_PS:	BOOL;
	STATE_OK:				BOOL;
END_VAR
VAR
	FM_ETAPE1:		R_TRIG;
	FM_ETAPE2:		R_TRIG;
	FM_ETAPE3:		R_TRIG;
	FM_ETAPE4:		R_TRIG;
	TIMER:					TON;
END_VAR

FM_ETAPE1(CLK:=OP_RUN.Etape.1);
FM_ETAPE2(CLK:=OP_RUN.Etape.2);
FM_ETAPE3(CLK:=OP_RUN.Etape.3);
FM_ETAPE4(CLK:=OP_RUN.Etape.4);


RQ_ROTATION_PS:= FM_ETAPE1.Q AND NOT I_NO_ROTATION_PS;
RQ_STOP_ROTATION_PS := (FM_ETAPE1.Q AND I_NO_ROTATION_PS) OR FM_ETAPE3.Q;

TIMER( PT:= DINT_TO_TIME(PRM_TIME*1000),
		IN:=OP_RUN.Etape.2);
		
STATE_OK := OP_RUN.OK;

RUN_STEP();

ACTION RUN_STEP:
(*GRAFCET ETAPE EFFLUVAGE*)
(* initialisation du grafcet*)
OP_RUN(
	N_STEP_OP_OK:=4 ,
	N_STEP_OP_NOK:= 0);

(* initialisation du grafcet*)
IF 		OP_RUN.Etape = 0 THEN
				OP_RUN.Etape.0 := TRUE;
(*repositionnement sur étape 0*)
ELSIF  NOT I_ON THEN
		OP_RUN.Etape:= 0;			(*RAZ grafcet*)
		OP_RUN.Etape.0:= TRUE;
(*étape 0-1 *)
ELSIF OP_RUN.Etape.0 AND I_ON  THEN
		OP_RUN.Etape.1 	:= TRUE;
		OP_RUN.Etape.0 	:= FALSE;
(*étape 2-1*)
ELSIF OP_RUN.Etape.1 AND ((I_ROTATION_OK AND NOT I_NO_ROTATION_PS) OR (I_STOP_ROT_PS_OK AND I_NO_ROTATION_PS)) THEN
		OP_RUN.Etape.2 	:= TRUE;
		OP_RUN.Etape.1 	:= FALSE;
(*étape 2-3*)
ELSIF OP_RUN.Etape.2 AND TIMER.Q THEN 
		OP_RUN.Etape.3	:= TRUE;
		OP_RUN.Etape.2	:= FALSE;
(*étape 3-4*)
ELSIF OP_RUN.Etape.3 AND I_STOP_ROT_PS_OK THEN 
		OP_RUN.Etape.4	:= TRUE;
		OP_RUN.Etape.3	:= FALSE;
END_IF

OP_RUN.POST();
END_ACTION

END_FUNCTION_BLOCK

// ---- POUs/FONCTION DE BASE/BLOCK_G7.TcPOU
FUNCTION_BLOCK BLOCK_G7

(* Fonction de gestion d'un G7 standard*)

(****************historique des versions*****************************)

(* Version 1-0 - ?? - VERSION INIITIALE - 15/02/2010*)
(* Verstion 1.1 - SP - Rationnalisation du bloc *)
(*************************************************************************)


VAR_INPUT
	N_STEP_OP_OK:				UINT (0..31);				(*n° d'étape correspondant à l'état OPERATION OK - 0 = inhibé*)
	N_STEP_OP_NOK:				UINT (0..31);				(*n° d'étape correspondant à l'état OPERATION NOK - 0 = inhibé*)
	OK:							BOOL;					(*code d'état OK de l'opération*)
	EC:							BOOL;					(*code d'état EN COURS de l'opération*)
	AR:							BOOL;					(*code d'état de l'opération à l'ARRET*)
	NOK:						BOOL;					(*code d'état de l'opération Non OK*)
	Etape:						UDINT;					(*étape du grafcet*)
END_VAR

VAR_OUTPUT
	STATUS:						UINT;	(* ~ (OPC : 1 : available for OPC-clients) *)				(*code d'état de l'opération*)
END_VAR

RETURN;

ACTION POST:
(*renvoi du code d'état de l'opération*)
STATUS 	:= 		LREAL_TO_UINT(LN(UDINT_TO_REAL(etape)) / LN(2));

(*drapeau d'état de la fonction*)
OK		:=		(ETAPE=EXPT(2,N_STEP_OP_OK)) AND (N_STEP_OP_OK>0);
AR		:=		ETAPE.0;
EC 		:= 		NOT OK AND NOT AR;
NOK		:=		(ETAPE=EXPT(2,N_STEP_OP_NOK)) AND (N_STEP_OP_NOK>0);
END_ACTION

END_FUNCTION_BLOCK

// ---- POUs/Fonction/FONCTION MODEMARCHE/BLOCK_STEP_EFFLUVAGE.TcPOU
FUNCTION_BLOCK BLOCK_STEP_EFFLUVAGE

(* Gestion etape d'effluvage avec injection de gaz par vanne microfuite*)

(****************historique des versions*****************************)

(* Version 0-0 - GV - VERSION INITIALE EVA760 n°113 - 9070*)
(* Version 1-0 - GV - VERSION EVA760 n°119 - 13375 - Modification pour gestion avec 2 lignes de gaz *)

(*************************************************************************)

VAR_INPUT
	I_ON:							BOOL;					(*Condition de déclenchement du grafcet d'étape d'effluvage*)
	I_POMPAGE_PRIM_OK:				BOOL;					(*Condition de pompage primaire ok*)
	I_POMPAGE_SEC_OK:				BOOL;					(*Condition pompage secondaire ok*)
	I_ROTATION_OK:					BOOL;					(*Condition rotation ok*)
	I_STOP_ROT_PS_OK:				BOOL;					(*Retour rotation PS à l'arrêt*)
	I_NO_ROTATION_PS:				BOOL;					(*Pas de rotation PS si consigne nulle*)
	I_ISOLEMENT_OK:					BOOL;					(*Condition isolement ok*)
	I_MARCHE_GAZ1_OK:				BOOL;					(*Mise en gaz ligne 1 ok*)
	I_ARRET_GAZ1_OK:				BOOL;					(*Arret gaz ligne 1 ok*)
	I_MARCHE_GAZ2_OK:				BOOL;					(*Mise en gaz ligne 2 ok*)
	I_ARRET_GAZ2_OK:				BOOL;					(*Arret gaz ligne 2 ok*)
	I_MARCHE_EFFLUVAGE_OK:			BOOL;					(*Retour effluvage ok*)
	I_ARRET_EFFLUVAGE_OK:			BOOL;					(*Retour arret effluvage ok*)
	TH_PPRIM_AUTOR:					BOOL;					(*Pression d'autorisation de pompage primaire atteinte*)
	TH_EFFLUVAGE:					BOOL;					(*Seuil de vide avant effluvage*)
	OP_RUN:							BLOCK_G7;				(*Grafcet de gestion de l'execution procede*)
	I_MODE_REPRISE:					BOOL;					(*indicateur de mode reprise en cours*)
	M_NEXT_STEP:					BOOL;					(*Demande externe de passage à l'étape suivante*)
	DEF_SEUIL_POMPAGE_PRIM: 		PRCDEF;				(*Défaut d'obtention du seuil de pompage primaire*)
	DEF_SEUIL_VIDE_EFFLUVAGE:		PRCDEF;				(*Défaut d'obtention du seuil de vide avant effluvage*)
	
	PRM_FLOW_GAZ1:				REAL;					(*Consigne de débit de gaz ligne 1*)
	PRM_FLOW_GAZ2:				REAL;					(*Consigne de débit de gaz ligne 2*)
END_VAR

VAR_INPUT PERSISTENT
	PRM_PR_EFFLUVAGE:			REAL;				(*Pression d'effluvage*)
	PRM_TEMPS_EFF:				TIME;				(*Temps de l'étape d'effluvage*)
	PRM_TPS_STABILISATION:		DINT;				(*Temps de stabilisation avant effluvage*)

	IsFunction:		BOOL;			(*entité : fonction*)
	IdXML:			STRING;			(*nom entité : identifiant pour recherche dans dico*)
	TagXML:			UINT;			(*nom entité : identifiant pour recherche dans dico*)
	IdParent:		STRING;			(*MNEMO de l'appelant*)
	MNEMO:			STRING;			(*MNEMO de l'entité*)
END_VAR

VAR_OUTPUT
	RQ_POMPAGE_PRIM:				BOOL;					(*Demande de pompage primaire*)
	RQ_POMPAGE_SEC:					BOOL;					(*Demande de pompage secondaire*)
	RQ_ISOLEMENT:					BOOL;					(*Demande d'isolement de l'enceinte*)
	RQ_MARCHE_GAZ:					ARRAY[0..2] OF BOOL;	(*Demande marche des lignes de gaz*)
	RQ_ARRET_GAZ:					BOOL;					(*Demande arrêt des lignes de gaz*)
	RQ_MARCHE_EFFLUVAGE:			BOOL;
	RQ_ARRET_EFFLUVAGE:				BOOL;
	RQ_ROTATION_PS:					BOOL;
	RQ_STOP_ROTATION_PS:			BOOL;
	STATE_OK:						BOOL;
	STATUS:							UINT;					(*Etat du grafcet*)
	AUTOR_NEXT_STEP:				BOOL;
END_VAR

VAR_IN_OUT
	CONS_TPS_EFFLUVAGE:				TIME;
	
	CONS_FLOW_GAZ_1:			REAL;	(*Consigne de débit de la mise en gaz*)
	CONS_FLOW_GAZ_2:			REAL;	(*Consigne de débit de la mise en gaz*)
END_VAR
VAR
	FM_ETAPE1:		R_TRIG;
	FM_ETAPE2:		R_TRIG;
	FM_ETAPE3:		R_TRIG;
	FM_ETAPE4:		R_TRIG;
	FM_ETAPE5:		R_TRIG;
	FM_ETAPE6:		R_TRIG;
	FM_ETAPE7:		R_TRIG;
	FM_ETAPE8:		R_TRIG;
	FM_ETAPE9:		R_TRIG;
	FM_ETAPE11:		R_TRIG;
	RCP_NEXT_STEP:	BOOL;
	TIMER_Stabilisation:			TON;			(*Temporisation de stabilisation*)
	
	VAR_Util_Gaz:					ARRAY[0..2] OF BOOL;		(*Indicateur des lignes de gaz utilisées*)
END_VAR

DEF_SEUIL_POMPAGE_PRIM.IdXML := '1';
DEF_SEUIL_POMPAGE_PRIM.TagXML := 24;

DEF_SEUIL_VIDE_EFFLUVAGE.IdXML := '1';
DEF_SEUIL_VIDE_EFFLUVAGE.TagXML := 25;

IdXML :='19';
TagXML := 4;

(*Reception des ordres*)
RCP_NEXT_STEP:= M_NEXT_STEP;

FM_ETAPE1(CLK:=OP_RUN.Etape.1);
FM_ETAPE2(CLK:=OP_RUN.Etape.2);
FM_ETAPE3(CLK:=OP_RUN.Etape.3);
FM_ETAPE4(CLK:=OP_RUN.Etape.4);
FM_ETAPE5(CLK:=OP_RUN.Etape.5);
FM_ETAPE6(CLK:=OP_RUN.Etape.6);
FM_ETAPE7(CLK:=OP_RUN.Etape.7);
FM_ETAPE8(CLK:=OP_RUN.Etape.8);
FM_ETAPE9(CLK:=OP_RUN.Etape.9);
FM_ETAPE11(CLK:=OP_RUN.Etape.11);


AUTOR_NEXT_STEP		:=	OP_RUN.Etape.1 OR OP_RUN.Etape.2 OR OP_RUN.Etape.3 OR OP_RUN.Etape.4 OR OP_RUN.Etape.5 OR OP_RUN.Etape.6 OR OP_RUN.Etape.7 OR OP_RUN.Etape.11;

(*Variable indiquant les lignes de gaz utilisées*)
VAR_Util_Gaz[1]:= (PRM_FLOW_GAZ1 > 0);
VAR_Util_Gaz[2]:= (PRM_FLOW_GAZ2 > 0);


RQ_POMPAGE_PRIM:= FM_ETAPE11.Q;
RQ_POMPAGE_SEC:= FM_ETAPE9.Q;
RQ_MARCHE_GAZ[1]:= (OP_RUN.Etape.3 OR OP_RUN.Etape.5) AND VAR_Util_Gaz[1];
RQ_MARCHE_GAZ[2]:= (OP_RUN.Etape.3 OR OP_RUN.Etape.5) AND VAR_Util_Gaz[2];
RQ_ISOLEMENT:=FM_ETAPE2.Q;
RQ_ROTATION_PS:= FM_ETAPE6.Q AND NOT I_NO_ROTATION_PS;
RQ_STOP_ROTATION_PS := (FM_ETAPE6.Q AND I_NO_ROTATION_PS) OR FM_ETAPE8.Q;
RQ_MARCHE_EFFLUVAGE:=FM_ETAPE7.Q;
RQ_ARRET_EFFLUVAGE:=FM_ETAPE8.Q;

RQ_ARRET_GAZ:= FM_ETAPE4.Q OR FM_ETAPE8.Q;

IF FM_ETAPE7.Q THEN
	CONS_TPS_EFFLUVAGE := PRM_TEMPS_EFF;
END_IF

(*Gestion de la consigne pour la ligne de gaz n°1*)
IF RQ_MARCHE_GAZ[1] THEN
	CONS_FLOW_GAZ_1 := PRM_FLOW_GAZ1;
END_IF

(*Gestion de la consigne pour la ligne de gaz n°2*)
IF RQ_MARCHE_GAZ[2] THEN
	CONS_FLOW_GAZ_2 := PRM_FLOW_GAZ2;
END_IF

(*Tempo de stabilisation de la pression*)
TIMER_Stabilisation(
					PT:=DINT_TO_TIME(PRM_TPS_STABILISATION*1000),
					IN:=OP_RUN.Etape.6
					);

(*Défaut obtention seuil pompage primaire*)
DEF_Seuil_Pompage_prim(
	CONDITION:= OP_RUN.Etape.3,
	DELAY:= T#3m);

(*Défaut obtention seuil de vide avant effluvage*)
DEF_Seuil_Vide_Effluvage(
	CONDITION:= OP_RUN.Etape.11,
	DELAY:= T#3m);


STATE_OK:=OP_RUN.OK;
STATUS:=OP_RUN.STATUS ;

RUN_STEP();

(*reset des ordres*)
IF RCP_NEXT_STEP AND M_NEXT_STEP THEN
	M_NEXT_STEP:=FALSE;
END_IF;

ACTION RUN_STEP:
(*GRAFCET ETAPE EFFLUVAGE*)
(* initialisation du grafcet*)
OP_RUN(
	N_STEP_OP_OK:=10 ,
	N_STEP_OP_NOK:= 0);

(* initialisation du grafcet*)
IF 		OP_RUN.Etape = 0 THEN
				OP_RUN.Etape.0 := TRUE;
(*interruption du procédé - repositionnement sur étape 8 sur demande fin d'étape*)
ELSIF (OP_RUN.Etape.1 OR OP_RUN.Etape.2 OR OP_RUN.Etape.3 OR OP_RUN.Etape.4 OR OP_RUN.Etape.5 OR OP_RUN.Etape.6 OR OP_RUN.Etape.7 OR OP_RUN.Etape.11)
		AND RCP_NEXT_STEP THEN
				OP_RUN.Etape := 0;
				OP_RUN.Etape.8:=TRUE;
(*repositionnement sur étape 0*)
ELSIF  NOT I_ON THEN
				OP_Run.Etape:= 0;			(*RAZ grafcet*)
				OP_Run.Etape.0:=TRUE;
(*étape 0-1 *)
ELSIF OP_RUN.etape.0 AND I_ON  THEN
				OP_RUN.Etape.1 	:=TRUE;
				OP_RUN.Etape.0 	:=FALSE;
(*étape 1-2*)
ELSIF OP_RUN.etape.1 AND NOT TH_PPRIM_AUTOR THEN		(*Pression < Pression autorisation pompage primaire*)
				OP_RUN.Etape.2 	:=TRUE;
				OP_RUN.Etape.1 	:=FALSE;
(*étape 1-4*)
ELSIF OP_RUN.etape.1 AND TH_PPRIM_AUTOR THEN
				OP_RUN.Etape.4 	:=TRUE;
				OP_RUN.Etape.1 	:=FALSE;
(*étape 2-3*)
ELSIF OP_RUN.etape.2 AND I_ISOLEMENT_OK  THEN
				OP_RUN.Etape.3 	:=TRUE;
				OP_RUN.Etape.2 	:=FALSE;
(*étape 3-4*)
ELSIF OP_RUN.etape.3 AND (I_MARCHE_GAZ1_OK OR NOT VAR_Util_Gaz[1]) AND (I_MARCHE_GAZ2_OK OR NOT VAR_Util_Gaz[2]) AND TH_PPRIM_AUTOR  THEN
				OP_RUN.Etape.4 	:=TRUE;
				OP_RUN.Etape.3 	:=FALSE;
(*étape 4-11*)
ELSIF OP_RUN.Etape.4 AND I_ARRET_GAZ1_OK AND I_ARRET_GAZ2_OK THEN
				OP_RUN.Etape.11 :=TRUE;
				OP_RUN.Etape.4	 := FALSE;
(*étape 11-5*)
ELSIF OP_RUN.etape.11 AND I_POMPAGE_PRIM_OK AND TH_EFFLUVAGE  THEN
				OP_RUN.Etape.5 	:=TRUE;
				OP_RUN.Etape.11:=FALSE;
(*étape 5-6*)
ELSIF OP_RUN.etape.5 AND (I_MARCHE_GAZ1_OK OR NOT VAR_Util_Gaz[1]) AND (I_MARCHE_GAZ2_OK OR NOT VAR_Util_Gaz[2]) THEN
				OP_RUN.Etape.6 	:=TRUE;
				OP_RUN.Etape.5 	:=FALSE;
(*étape 6-7*)
ELSIF OP_RUN.etape.6 AND TIMER_Stabilisation.Q
					  AND ((I_ROTATION_OK AND NOT I_NO_ROTATION_PS) OR (I_STOP_ROT_PS_OK AND I_NO_ROTATION_PS))
					  THEN
				OP_RUN.Etape.7 	:=TRUE;
				OP_RUN.Etape.6 	:=FALSE;
(*étape 7-8*)
ELSIF OP_RUN.etape.7 AND I_MARCHE_EFFLUVAGE_OK   THEN
				OP_RUN.Etape.8 	:=TRUE;
				OP_RUN.Etape.7 	:=FALSE;
(*étape 8-9*)
ELSIF OP_RUN.etape.8 AND I_ARRET_EFFLUVAGE_OK AND I_STOP_ROT_PS_OK AND I_ARRET_GAZ1_OK AND I_ARRET_GAZ2_OK THEN
				OP_RUN.Etape.9 	:=TRUE;
				OP_RUN.Etape.8 	:=FALSE;
(*étape 9-10*)
ELSIF OP_RUN.etape.9 AND I_POMPAGE_SEC_OK   THEN
				OP_RUN.Etape.10 :=TRUE;
				OP_RUN.Etape.9 	 :=FALSE;
END_IF

OP_RUN.POST();
END_ACTION

END_FUNCTION_BLOCK

// ---- POUs/FONCTION DE BASE/PRCDEF.TcPOU
FUNCTION_BLOCK PRCDEF

(* Fonction standard AC de gestion de défaut *)

(****************historique des versions*****************************)

(* Version 1-0 - SP - VERSION INIITIALE*)
(* Version 2-0 - HG - Adaptation pour journal des évènements externe - 24/06/2011*)

(*************************************************************************)


VAR_INPUT
	CONDITION:	  				BOOL;				(* ~ (OPC : 1 : available for OPC-clients) *)			(*condition d'apparition du défaut*)
	DISABLE:					BOOL:=FALSE;													(*condition de désactivation du défaut*)
	AR_DEF:   					BOOL:=TRUE; 		(* ~ (OPC : 1 : available for OPC-clients) *)			(* Accusé de reception du défaut *)
END_VAR

VAR_INPUT PERSISTENT
	DELAY:		  				TIME;		 		(* ~ (OPC : 1 : available for OPC-clients) *)			(* Delais du défaut pour l'obtention de la réaction*)
	COUNT_APP:				UDINT;				(* ~ (OPC : 1 : available for OPC-clients) *)			(* Nombre d'apparition du défaut*)

	(*Entité*)
	IdXML:			STRING;			(*nom entité : identifiant pour recherche dans dico*)
	TagXML:			UINT;			(*nom entité : identifiant pour recherche dans dico*)
	Groupe:			UINT:=0;			(*0:defaut, 1:alarme, 2:utilisateur, 3:évènement, 4:consignation, 5:note*)
	VAL1:			STRING(255);		(*attribut pour affichage intitulé*)
	VAL2:			STRING;			(*attribut pour affichage intitulé*)
	VAL3:			STRING;			(*attribut pour affichage intitulé*)
	ID:				UINT;			(*identifiant du défaut*)
END_VAR

VAR_OUTPUT
	DEF:   						BOOL; 															(* indicateur de défaut *)
	APP	:						BOOL;															(* bit activé à l'apparition du défaut*)
	DIS:							BOOL;															(* bit activé à la disparition du défaut*)
END_VAR

VAR
	T_delay:						TON;															(*timer délais défaut*)
	FM_DEF:					R_TRIG;															(*APP du défaut*)
	FD_DEF:						F_TRIG;															(*DIS du défaut*)
	TIMER_AR:					TON;															(*Timer pour accusé de réception du délais de défaut*)
END_VAR

	T_DELAY.IN:= CONDITION AND NOT DISABLE;
	T_delay(	PT:=DELAY);

	TIMER_AR.PT	:=	T#5s;
	TIMER_AR.IN	:=	DEF;
	TIMER_AR();

	(************************************************************************************************)
	(* TRAITEMENT DES DEFAUTS AVEC DELAIS = 0 (APPARITION IMMEDIATE) *)
	(************************************************************************************************)

	IF		DELAY = T#0s THEN				 (* [Delais<>0] *)

		(* mis à 1 du défaut si la condition est vraie *)
		IF		CONDITION AND NOT DISABLE THEN
			DEF:=TRUE;
		END_IF;

	(* RAZ du defaut si pas condition *)
		IF (NOT CONDITION AND DEF AND AR_DEF) OR	DISABLE THEN
			DEF := FALSE;
		END_IF;

		(*TODO - A SHUNTER SI JEV OK*)
		IF (NOT CONDITION AND DEF  AND TIMER_AR.Q ) OR	DISABLE THEN
			DEF := FALSE;
		END_IF;
	ELSE
	(************************************************************************************************)
	(* TRAITEMENT DES DEFAUT AVEC DELAIS > 0                                                            *)
	(************************************************************************************************)

		IF T_delay.Q THEN
			DEF := TRUE;
		END_IF;
		IF	(DEF  AND AR_DEF AND NOT CONDITION) OR DISABLE THEN
				DEF:=FALSE;
		END_IF;
		(*TODO - A SHUNTER SI JEV OK*)
		IF	(DEF  AND TIMER_AR.Q AND NOT CONDITION) OR DISABLE THEN
				DEF:=FALSE;
		END_IF;
	END_IF;


	FM_DEF(CLK:=DEF , Q=>APP );
	FD_DEF(CLK:=DEF , Q=>DIS );

	IF APP THEN
		COUNT_APP:=COUNT_APP+1;
		LOG_EVENT(
			_ID:=ID,
			_VAL1:=VAL1,
			_VAL2:=VAL2,
			_VAL3:=VAL3,
			_TYPE:=TRUE);

	END_IF;
	IF DIS THEN
			LOG_EVENT(
			_ID:=ID,
			_VAL1:=VAL1,
			_VAL2:=VAL2,
			_VAL3:=VAL3,
			_TYPE:=FALSE);
	END_IF
	IF ID < SIZEOF(PRG_DEF_MANAGEMENT.TABLE_DEF) * 32 THEN
		 PRG_DEF_MANAGEMENT.TABLE_DEF[ ID / 32] := CSETBIT32(
			inVal32:= PRG_DEF_MANAGEMENT.TABLE_DEF[ ID / 32],
			BitNo:=UINT_TO_USINT( ID MOD 32),
			BitVal:= DEF);
	ELSE
			ADSLOGSTR(ADSLOG_MSGTYPE_ERROR,'indice de table de défaut dépassé', '');
	END_IF

END_FUNCTION_BLOCK

// ---- POUs/FONCTION DE BASE/LOG_EVENT.TcPOU
FUNCTION LOG_EVENT : BOOL
VAR_INPUT
	_ID:		UINT;	(*indentifiant du défaut*)
	_VAL1:	STRING;
	_VAL2:	STRING;
	_VAL3:	STRING;
	_TYPE:	BOOL;	(*0=disparition , 1= apparition*)
END_VAR
VAR
	I:	UINT;
END_VAR

	FOR I:=0 TO 99 DO
		IF PRG_DEF_MANAGEMENT.EVENT_MAILBOX[i]._ID = 0 THEN
			PRG_DEF_MANAGEMENT.EVENT_MAILBOX[i]._ID:=_ID;
			PRG_DEF_MANAGEMENT.EVENT_MAILBOX[i]._VAL1:=_VAL1;
			PRG_DEF_MANAGEMENT.EVENT_MAILBOX[i]._VAL2:=_VAL2;
			PRG_DEF_MANAGEMENT.EVENT_MAILBOX[i]._VAL3:=_VAL3;
			PRG_DEF_MANAGEMENT.EVENT_MAILBOX[i]._TYPE:=_TYPE;
			PRG_DEF_MANAGEMENT.EVENT_MAILBOX[i]._HORODAT:= PRG_SEC._date;
			PRG_DEF_MANAGEMENT.EVENT_MAILBOX[i]._MS:=PRG_SEC._ms;
			EXIT;
		END_IF
		(*PRG_DEF_MANAGEMENT.EVENT_MAILBOX_FULL;*)
	END_FOR

END_FUNCTION

// ---- POUs/Programme/PRG_DEF_MANAGEMENT.TcPOU
PROGRAM PRG_DEF_MANAGEMENT
(* V1.0 S.PARISOT 01/2012 Gestion des piles de défaut et de la communication avec ACsoft*)
VAR_OUTPUT
	EVENT_MAILBOX_FULL:	BOOL;
	STATE_DEFAUT_PRESENT:	BOOL;		(*Indicateur de défaut en cours sur équipement, levé par journal externe*)
END_VAR
VAR_INPUT
	RQ_EMPTY:				BOOL;								(*demande de vidage de la pile*)
	TABLE_DEF:				ARRAY[0..30] OF DWORD;				(*tables d'état des défaut - 960 defaut max*)
	RQ_DISPLAY_EVENT:		BOOL;								(*demande d'enregistrement d'un événement dans la liste des événements récents*)
END_VAR
VAR_INPUT PERSISTENT
	EVENT_MAILBOX:		ARRAY[0..100] OF STRUCT_EVENT;	(* pile des evenements en attente de prise en compte par le module EVENT*)
	EVENT_LIST:			ARRAY[0..20] OF STRUCT_JEV;		(*Liste des événements récents pour affichage dans l'IHM*)
	EVENT_TO_SEND:		STRUCT_EVENT;					(*Evenement en attente d'enregistrement dans la base de donnée*)
	EVENT_TO_DISPLAY:	STRUCT_JEV;						(*Evenement en attente d'enregistrement dans la liste des événements récents*)
END_VAR

VAR
	I:	INT;
END_VAR

(* le module AC-SOFTWARE demande l'affichage de l'évenement dans la table des événements récents*)
IF RQ_DISPLAY_EVENT THEN
	I:=19;
	WHILE (i>=0) DO
		EVENT_LIST[I+1] := EVENT_LIST[I];
		I:=I-1;
	END_WHILE
	EVENT_LIST[0] := EVENT_TO_DISPLAY;
	RQ_DISPLAY_EVENT:= FALSE;

END_IF
(* si l'id de l'évenement à envoyer est = 0 (pas d'evenement dans la boite) alors*)
IF  (EVENT_TO_SEND._ID = 0) THEN
	(* si le premier evenement de la pile d'évenement n'est pas nulle (= présence d'un évenement en haut  de la pile) *)
	IF NOT (EVENT_MAILBOX[0]._ID = 0) THEN
		(*on informe le type et l'horodatage de l'événement en attente d'ebregistrement dans la liste des événements récents*)
		IF EVENT_MAILBOX[0]._TYPE  THEN
			EVENT_TO_DISPLAY.STATE_App := 'APP';
		ELSE
			EVENT_TO_DISPLAY.STATE_App := 'DIS';
		END_IF
		EVENT_TO_DISPLAY.STATE_DT := EVENT_MAILBOX[0]._HORODAT;
	END_IF
	(*on met l'évenement en haut de  la pile en attente d'envoi vers la base de donnée *)
	EVENT_TO_SEND:=EVENT_MAILBOX[0];
	(*on décale toute la pile vers le haut*)
	FOR i:=0 TO 99 DO
		EVENT_MAILBOX[i]:=EVENT_MAILBOX[i+1];
		EVENT_MAILBOX[100]._ID := 0;
	END_FOR

END_IF


IF RQ_EMPTY THEN
FOR i:=0 TO 99 DO
		EVENT_TO_SEND._ID := 0;
		EVENT_MAILBOX[i]._ID := 0;
END_FOR
END_IF

END_PROGRAM

// ---- POUs/Fonction/FONCTION EVAPORATION/BLOCK_STEP_EMPILEMENT.TcPOU
FUNCTION_BLOCK BLOCK_STEP_EMPILEMENT

(* Gestion empilement de couche *)

(****************historique des versions*****************************)

(* Version 0-0 - SD - VERSION INITIALE CT200 n°7 - 8157 *)
(* Version 1-0 - GV - Correction du bloc : - Pas de RAZ XTC sur reprise,
								    - Gestion fin de couche VAR_MEM_COUCHE_TERMINEE
								    - Pas de rechargement des paramètres XTC sur reprise 
								    - Pas de répition des boucles si couche suivante
								    - ...*)
(* Version 2-0 - GV - Pas de demande de rotation PS si consigne nulle (Etape 6) - 06/2015 - 8866 *)
(* Version 3-0 - GV - Gestion introduction gaz et regulation de pression - 07/2015 - 9070 *)
(* Version 4-0 - GV - Ajout gestion de demande de tilt PS + Modification gestion IAD + Modification gestion chauffage*)
(* Version 5-0 - HG - Ajout option condition gaz/pression pour chaque segment avec application des conditions de gaz et pression si oui, pompage secondaire sans gaz sinon*)
(* Version 6-0 - GV - Ajout d'un evenement épaisseur déposée en fin de couche*)
(* Version 6-1 - GV - Correction Reset VAR_Cond_MGaz sur Etape 1*)

(*************************************************************************)

VAR_INPUT
	I_ON:							BOOL;					(*Condition de déclenchement du grafcet de marche du procédé*)

	I_LAYER_LOADING_OK:				BOOL;					(*L'IHM indique le chargement de la couche ok*)
	I_LAYER_LOADING_NOK:			BOOL;					(*L'IHM indique le chargement de la couche nok*)

	I_LAYER_ANT_LOADING_OK:			BOOL;					(*chargement de la couche anticipée Ok*)
	I_LAYER_ANT_LOADING_NOK:		BOOL;					(*chargement de la couche anticipée NOk*)

	I_NO_MORE_LAYER:				BOOL;					(*L'IHM indique qu'il n'y a plus de couche à exécuter*)
	I_NO_MORE_LAYER_ANT:			BOOL;					(*plus de couche anticipée à lancer*)

(*	I_STEP_NUMBER:				UINT;				(*Numéro de l'étape dans l'empilement*)	*)

	I_ACTION_CONTROLEUR_OK:		BOOL;				(*Retour action contrôleur OK, RESET,RAZ,STOP etc*)
	I_CONTROLEUR_PHASE:			STRING;				(*Etat du contrôleur *)

	I_PROG_CONTROLEUR_OK:			BOOL;				(*Retour programmation contrôleur OK*)
	I_END_DEPOT:					BOOL;				(*Retour indiquant que le dépôt est terminé*)

	I_STAB_CHAUFFAGE_OK:			BOOL;				(*Stabilisation chauffage ok*)
	I_CONTROLEUR_STOPPED:			BOOL;				(*Retour contrôleur de depôt à l'arrêt*)

	I_N_SEGMENT_S1:				USINT;				(*N° de segment en cours pour la source 1*)
	I_N_SEGMENT_S2:				USINT;				(*N° de segment en cours pour la source 2*)
	I_N_SEGMENT_S3:				USINT;				(*N° de segment en cours pour la source 3*)
	I_N_SEGMENT_S4:				USINT;				(*N° de segment en cours pour la source 4*)

	CONF_CHAUFFAGE:					BOOL;				(*Indique s'il y a du chauffage*)
	CONF_IAD:						BOOL;				(*Indique s'il y a un IAD*)

	I_ROTATION_PS_OK:				BOOL;				(*Retour rotation PS ok*)
	I_TILT_PS_OK:					BOOL;				(*Retour tilt PS ok*)
	I_STOP_ROT_PS_OK:				BOOL;				(*Retour rotation PS à l'arrêt*)
	I_STOP_TILT_PS_OK:				BOOL;				(*Retour tilt PS à l'arrêt*)
	I_NO_ROTATION_PS:				BOOL;				(*Pas de rotation PS si consigne nulle*)
	I_MODE_TILT:					INT;					(*Retour de sélection mode tilt (1: Balayage, 2: Position)*)
	I_MARCHE_CHAUFFAGE_OK:			BOOL;				(*Retour marche Chauffage PS ok*)
	I_ARRET_CHAUFFAGE_OK:			BOOL;				(*Retour Arrêt chauffage ok*)
	I_MARCHE_GAZ1_OK:				BOOL;				(*Retour marche gaz 1 ok*)
	I_MARCHE_GAZ2_OK:				BOOL;				(*Retour marche gaz 2 ok*)
	I_ARRET_GAZ1_OK:				BOOL;				(*Retour Arrêt gaz 1 ok*)
	I_ARRET_GAZ2_OK:				BOOL;				(*Retour Arrêt gaz 2 ok*)
	I_ARRET_REGUL_GAZ_OK:		ARRAY[0..2] OF BOOL;(*Retour arrêt regulation de pression en débit de gaz*)
	I_MARCHE_POMPAGE_PROC_OK:	BOOL;				(*Retour pompage procédé ok*)
	I_MARCHE_POMPAGE_SEC_OK:	BOOL;				(*Retour pompage secondaire ok*)
	I_MARCHE_IAD_OK:				BOOL;				(*Retour marche IAD OK*)
	I_ARRET_IAD_OK:					BOOL;				(*Retour arrêt IAD OK*)
	I_POSITIONNEMENT_OK:			BOOL;				(*Retour positionnement de l'axe Z OK*)

	I_PREP_SOURCE1_OK:			BOOL;				(*Retour préparation source 1 ok*)
	I_PREP_SOURCE2_OK:			BOOL;				(*Retour préparation source 2 ok*)
	I_PREP_SOURCE3_OK:			BOOL;				(*Retour préparation source 3 ok*)
	I_PREP_SOURCE4_OK:			BOOL;				(*Retour préparation source 4 ok*)

	I_EVAP1_OK:						BOOL;				(*Source 1 en phase d'évaporation*)
	I_EVAP2_OK:						BOOL;				(*Source 2 en phase d'évaporation*)
	I_EVAP3_OK:						BOOL;				(*Source 3 en phase d'évaporation*)
	I_EVAP4_OK:						BOOL;				(*Source 4 en phase d'évaporation*)

	I_SOURCE1_PREFU:				BOOL;				(*Retour source 1 en préparation, phase de préfusion*)
	I_SOURCE2_PREFU:				BOOL;				(*Retour source 2 en préparation, phase de préfusion*)
	I_SOURCE3_PREFU:				BOOL;				(*Retour source 3 en préparation, phase de préfusion*)
	I_SOURCE4_PREFU:				BOOL;				(*Retour source 4 en préparation, phase de préfusion*)

	I_SOURCE1_IDLE:				BOOL;				(*Retour source 1 en IDLE*)
	I_SOURCE2_IDLE:				BOOL;				(*Retour source 2 en IDLE*)
	I_SOURCE3_IDLE:				BOOL;				(*Retour source 3 en IDLE*)
	I_SOURCE4_IDLE:				BOOL;				(*Retour source 4 en IDLE*)

	I_CLOT_SOURCE1_OK:			BOOL;				(*Cloture de la source 1 ok*)
	I_CLOT_SOURCE2_OK:			BOOL;				(*Cloture de la source 2 ok*)
	I_CLOT_SOURCE3_OK:			BOOL;				(*Cloture de la source 3 ok*)
	I_CLOT_SOURCE4_OK:			BOOL;				(*Cloture de la source 4 ok*)

	I_STOP_EVAP1_OK:				BOOL;				(*Source 1 à l'arrêt*)
	I_STOP_EVAP2_OK:				BOOL;				(*Source 2 à l'arrêt*)
	I_STOP_EVAP3_OK:				BOOL;				(*Source 3 à l'arrêt*)
	I_STOP_EVAP4_OK:				BOOL;				(*Source 4 à l'arrêt*)

	M_NEXT_LAYER:					BOOL;				(*IHM demande le passage à la couche suivante*)
	PRM_OP_UTIL_IAD:				BOOL;				(*Parametre indiquant l'utilisation d'un IAD*)

	I_DOME_IN_POSITION:			BOOL;		(*Indique si le dome est en position*)

(*Vitesse/Epaisseur de dépôt global*)
	I_Global_Thick:					REAL;
	I_Global_Rate:					REAL;

(*Indique si la source est arrêté ou sa cloture est terminée*)
	I_SOURCE1_ARRET:				BOOL;
	I_SOURCE2_ARRET:				BOOL;
	I_SOURCE3_ARRET:				BOOL;
	I_SOURCE4_ARRET:				BOOL;

(*Temps de préparation des sources*)
	PRM_TPS_PREPA_SOURCE1:		INT;
	PRM_TPS_PREPA_SOURCE2:		INT;
	PRM_TPS_PREPA_SOURCE3:		INT;
	PRM_TPS_PREPA_SOURCE4:		INT;
(*Vitesse d'évaporation théorique des sources*)
	PRM_SOURCE1_RATE:			REAL;
	PRM_SOURCE2_RATE:			REAL;
	PRM_SOURCE3_RATE:			REAL;
	PRM_SOURCE4_RATE:			REAL;

(*Parametres indiquant s'il y a utilisation d'un quartz pour l'étalonnage*)
	PRM_CTRL_DELAY_SOURCE1:	BOOL;
	PRM_CTRL_DELAY_SOURCE2:	BOOL;
	PRM_CTRL_DELAY_SOURCE3:	BOOL;
	PRM_CTRL_DELAY_SOURCE4:	BOOL;

(*sources utilisées pour couche en cours*)
	PRM_UTIL_SOURCE1:			BOOL;
	PRM_UTIL_SOURCE2:			BOOL;
	PRM_UTIL_SOURCE3:			BOOL;
	PRM_UTIL_SOURCE4:			BOOL;

(*sources utilisées pour couche anticipée*)
	PRM_UTIL_SOURCE1_ANT:		BOOL;
	PRM_UTIL_SOURCE2_ANT:		BOOL;
	PRM_UTIL_SOURCE3_ANT:		BOOL;
	PRM_UTIL_SOURCE4_ANT:		BOOL;

	PRM_MAIN_TOOLING:			REAL;	(*Facteur de correction global*)
	PRM_TOOLING_QZ:				ARRAY[0..11]OF REAL;		(*Facteur de correction de chaque Quartz*)
	PRM_POIDS_QZ:				ARRAY[0..11]OF REAL;		(*Paramêtres indiquant le poids de chaque quartz dans la mesure*)
	PRM_ZRATIO_QZ:				ARRAY[0..11]OF REAL;		(*Parametres indiquant le z-ratio afécté au quartz*)
	PRM_DENSITE_QZ:				ARRAY[0..11]OF REAL;		(*Densité affecté à chaque quartz*)
	PRM_TIMEPOWER:				BOOL;	(*Réaction en cas de panne du quartz associé au controle vitesse de la source
																						0 = arrêt de couche
																						1 = fin de la couche à la puissance moyenne
																						*)

	PRM_FACTEUR_FINE:			REAL;		(*Facteur de correction fine appliqué au tooling des Quartz*)

	(*Paramètre pompage procédé*)
	PRM_MODE_PUMPING:			USINT;		(*Option mode de régulation 0:position, 1:pression, 2:gaz 1, 3:gaz 2*)
	PRM_PR_PUMPING:				REAL;		(*Pression de regulation*)
	PRM_POS_PUMPING:			REAL;		(*Position vanne asservie*)
	PRM_PR_HI_PUMPING:			REAL;		(*Pression limite haute*)
	PRM_PR_LO_PUMPING:			REAL;		(*Pression limite basse*)
	PRM_TIM_PR_PUMPING:			REAL;		(*Temps stabilisation pression*)

	(**)
	PRM_MATERIAU_MACHINE:		STRING;		(*Nom du matériau machine (fiche matériau*)
	PRM_ANTICIPATION_COUCHE:	BOOL;		(*Indique que la couche en cours est anticipée (donc sa prépa a été lancée sur couche précédente)*)
	PRM_SOURCE_MAITRE:			USINT;
	PRM_EPAISSEUR:				REAL;		(*Epaisseur de dépôt à atteindre*)

	PRM_NEW_EPAISSEUR:			ARRAY[0..499] OF REAL;	 (*Nouvelles épaisseurs*)

	(*Paramètre de mise en gaz*)
	PRM_N_SEGMENT_GAZ:			INT;						(*N° de segment pour la mise en gaz*)
	PRM_FLOW_GAZ1:				REAL;					(*Consigne de débit de gaz ligne 1*)
	PRM_FLOW_GAZ2:				REAL;					(*Consigne de débit de gaz ligne 2*)
	PRM_GAZ_PRESSION_SEGMENT:	ARRAY[0..10] OF BOOL;	(*Option utilisation des conditions de gaz/pression indiquées pour le segment, sinon pompage secondaire sans gaz*)

	(*Paramètre de segment de chauffage*)
	PRM_MODE_CHAUFFAGE:			USINT;					(*mode chauffage*)
	PRM_WAIT_STAB_TEMP:			BOOL;					(*Attente stabilisation température*)
	PRM_TEMPERATURE:			REAL;					(*Consigne de température*)
	PRM_INC_RAMPE_CHAUFFAGE:	REAL;					(*en °C/min*)
	PRM_DELTA_TEMPERATURE:		REAL;					(*en °C*)
	PRM_TPS_STAB_TEMP:			REAL;					(*en min*)
	PRM_TPS_STAB_TEMP_MAX:		REAL;					(*en min*)

	(*Avance ouverture cache IAD*)
	PRM_AVANCE_IAD:				REAL;					(*Paramètres d'avance ouverture IAD*)

	(*défaut*)
	DEF_READ_LAYER:				PRCDEF;				(*défaut de lecture d'une étape*)
	DEF_READ_LAYER_ANT:			PRCDEF;				(*défaut de lecture d'une étape anticipée*)

	EV_LOAD_LAYER:				PRCDEF;				(*Evenement chargement d'une étape*)
	EV_NEXT_LAYER:				PRCDEF;				(*Evenement de passage à l'étape suivante*)
	EV_THICK_AGREGATE:			PRCDEF;				(*Evenement information épaisseur réel déposée*)
	DEF_RAZ_QZ:					PRCDEF;				(*Défaut de raz de l'épaisseur*)
	DEF_PROG_QZ:				PRCDEF;				(*Défaut de programmation de la couche*)
	DEF_QF:						PRCDEF;				(*Défaut de panne quartz générale - poids max atteint par un quartz*)
	DEF_CONTROLLER_STOPPED:		PRCDEF;				(*Défaut de passage en STOP du contrôleur de dépôt pendant l'évaporation*)

(*ajouté par seb*)
	(*DEF_SURV_TPS_DEPOT:		PRCDEF;			(*Défaut de surveillance du temps de dépôt*)*)
	EV_RELOAD:					PRCDEF;					(*Evenement de rechargement du programme*)

	OP_RUN:						BLOCK_G7;				(*Grafcet de gestion de l'execution procede*)


	PRM_QUARTZ_SOURCE:			BOOL;					(*indique si un quartz est présent sous le cache source*)


(*Parametre de boucle , définit s'il faut effectuer une repetition des couches*)
	PRM_LOOP:					BOOL;		(*Parametre indiquant s'il y a une boucle à effectuer*)
	PRM_LOOP_FIRST_LAYER:		UINT;		(*Numéro de début de la couche à répeter*)
	PRM_LOOP_LAST_LAYER:		UINT;		(*Numéro de fin de la couche à répeter*)
	PRM_NB_LOOP:				UINT;		(*Indique le nombre de repetition de la boucle*)


(*Parametre concernant le type de dôme selectionné dans le programme*)
	PRM_Type_Dome:				USINT;		(*0 =250mm, 1= 350mm, 2= 450mm*)


END_VAR
VAR_INPUT PERSISTENT
	IsFunction:						BOOL;			(*entité : fonction*)
	IdXML:							STRING;			(*nom entité : identifiant pour recherche dans dico*)
	TagXML:							UINT;			(*nom entité : identifiant pour recherche dans dico*)
	IdParent:						STRING;			(*MNEMO de l'appelant*)
	MNEMO:							STRING;			(*MNEMO de l'entité*)
	PRM_NQz_Min:					USINT:=1;		(*Nombre mini de quartz avant panne*)
	PRM_QF_Poids_Max: 				REAL;
	PRM_QF_VIE_Min:					REAL;
END_VAR
VAR_OUTPUT
	RQ_LOAD_PARAM:				BOOL;			(*Demande de chargement parametre Couche/Quartz dans le contrôleur de dépôt*)

	RQ_PREP_S1:					BOOL;			(*Demande de préparation de la source 1*)
	RQ_PREP_S2:					BOOL;			(*Demande de préparation de la source 2*)
	RQ_PREP_S3:					BOOL;			(*Demande de préparation de la source 3*)
	RQ_PREP_S4:					BOOL;			(*Demande de préparation de la source 4*)

	RQ_NEXT_LAYER:				BOOL;		(*Demande fin de couche*)

	RQ_EVAP_S1:					BOOL;				(*Demande de mise en phase évaporation de la source 1*)
	RQ_EVAP_S2:					BOOL;				(*Demande de mise en phase évaporation de la source 2*)
	RQ_EVAP_S3:					BOOL;				(*Demande de mise en phase évaporation de la source 3*)
	RQ_EVAP_S4:					BOOL;				(*Demande de mise en phase évaporation de la source 4*)

	RQ_ROTATION_PS:				BOOL;			(*Demande rotation PS*)
	RQ_TILT_PS:					BOOL;			(*Demande de tilt PS*)
	RQ_STOP_ROTATION_PS:		BOOL;			(*Demande Arrêt rotation PS*)
	RQ_STOP_TILT_PS:			BOOL;			(*Demande Arrêt tilt PS*)
	RQ_MARCHE_CHAUFFAGE:		BOOL;			(*Demande de marche du chauffage*)
	RQ_ARRET_CHAUFFAGE:			BOOL;			(*Demande d'arrêt du chauffage*)
	RQ_MARCHE_IAD:				BOOL;			(*Demande marche IAD*)
	RQ_ARRET_IAD:				BOOL;			(*Demande arrêt IAD*)

	RQ_POSITIONNEMENT_Z:		BOOL;			(*Demande de positionnement de l'axe Z*)

	RQ_MARCHE_GAZ:				ARRAY[0..2] OF BOOL;	(*Demande marche des lignes de gaz*)
	RQ_ARRET_GAZ:				ARRAY[0..2] OF BOOL;	(*Demande arrêt des lignes de gaz*)

	RQ_MARCHE_REGUL_GAZ:		ARRAY[0..2] OF BOOL;	(*Demande marche de la régulation en débit de gaz*)
	RQ_ARRET_REGUL_GAZ:			ARRAY[0..2] OF BOOL; 	(*Demande arrêt de la régulation en débit de gaz*)

	RQ_STOP_EVAP_S1:				BOOL;		(*Demande d'arrêt de la source 1*)
	RQ_STOP_EVAP_S2:				BOOL;		(*Demande d'arrêt de la source 2*)
	RQ_STOP_EVAP_S3:				BOOL;		(*Demande d'arrêt de la source 3*)
	RQ_STOP_EVAP_S4:				BOOL;		(*Demande d'arrêt de la source 4*)

	RQ_OUV_CC_Iad:					BOOL;		(*Demande ouverture cache IAD*)

	RQ_MARCHE_POMPAGE_PROC:	BOOL;		(*Demande de mise en pompage procédé*)
	RQ_MARCHE_POMPAGE_SEC:	BOOL;		(*Dempande de mise en pompage secondaire*)

	RQ_READ_LAYER:				BOOL;		(*Demande de lecture de l'étape suivante*)
	RQ_READ_LAYER_ANT:			BOOL;		(*Demande de lecture de la couche anticipée*)
(*	RQ_READ_NUM_LAYER:			BOOL;		(*Demande de lecture du numéro d'étape demandé*)
	OUT_NUM_LAYER_TO_READ:		UINT;		(*Indique le numéro de l'étape à lire*)
*)
	OUT_RAZ_THICK_CONTROLEUR:	BOOL;		(*Demande de RAZ epaisseur du contrôleur*)
	OUT_RESET_CONTROLEUR:		BOOL;		(*Demande de reset du controleur*)
	OUT_STOP_CONTROLEUR:		BOOL;		(*Demande d'arrêt du contrôleur*)

	STATE_OK:					BOOL;
	STATUS:						UINT;						(*Etat du grafcet*)
	STATE_LAYER:				UINT:=1;						(*N° de la couche en cours*)
	STATE_LAYER_TEXT:			STRING(255);					(*Descriptif de la couche en cours d'exécution*)
	AUTOR_NEXT_LAYER:			BOOL;
	STATE_RATE_AGREGATE:		REAL;						(*epaisseur globale*)
	STATE_THICKNESS_AGREGATE:	REAL;						(*Epaisseur globale*)
	VAR_MEM_RAZ_THICKNESS:		BOOL;						(*Mémorisation de la variable de remise à 0 de l'épaisseur*)
	TIMER_RAZ_THICKNESS:		TON;
	TIMER_RAZ_EPAISSEUR:		TON;

	STATE_END_OF_LAYER:			BOOL;		(*Indique que la couche en cours est terminée*)
	STATE_EVAP:					BOOL;		(*Indique que l'évaporation est en cours*)

	CONS_MODE:					USINT;	(*Consigne de mode de régulation de la pression*)
	CONS_PRESSURE:				REAL;	(*Consigne de pression en cas de regulation en pression*)
	CONS_POSITION:				REAL;	(*Consigne de position en cas de regulation en position*)
	CONS_HI_PRESSURE:			REAL;	(*Pression limite haute pour stabilisation*)
	CONS_LOW_PRESSURE:			REAL;	(*Pression limite basse pour stabilisation*)
	CONS_TIM_PRESSURE:			TIME;	(*Temps pour stabilisation pression*)

END_VAR

VAR_IN_OUT
	I_MODE_REPRISE:				BOOL;	(*information de mode reprise*)

	CONS_FLOW_GAZ_1:			REAL;	(*Consigne de débit de la mise en gaz*)
	CONS_FLOW_GAZ_2:			REAL;	(*Consigne de débit de la mise en gaz*)

	(*CONS_POSITION_DOME:		USINT;	(*Consigne de position du dôme*)*)
END_VAR

VAR
	TIMER_TIMEOUT:				TON;		(*Timer timemout lecture étape*)
	TIMER_TIMEOUT_ANT:			TON;		(*Timer timeout lecture étape anticipée*)

	RCP_NEXT_LAYER:				BOOL;
	FM_ETAPE20:					R_TRIG;
	FM_ETAPE6:					R_TRIG;
	FM_ETAPE7:					R_TRIG;
	FM_ETAPE9:					R_TRIG;
	FM_ETAPE10:					R_TRIG;
	FM_ETAPE11:					R_TRIG;
	FM_ETAPE12:					R_TRIG;
	FM_ETAPE13:					R_TRIG;
	FM_ETAPE14:					R_TRIG;
	FM_COND_MGAZ:				R_TRIG;		(*Condition de mise en gaz *)
	FD_COND_MGAZ:				F_TRIG;

	VAR_MEM_LAYER_INTERRUPTED:	BOOL;	(*mémoire de dépôt interrompue avant la fin de la couche*)
	VAR_MEM_COUCHE_TERMINEE:	BOOL;	(*mémoire de couche terminée - utiliser pour le mode reprise*)
	VAR_MEM_PREP_OPT_TERMINEE:	BOOL;	(*Mémoire de préparation optique terminée*)

	VAR_TPS_PREPA_ANT1:				INT;			(*calcul du temps nécessaire pour préparation des sources anticipées en secondes*)
	VAR_TPS_PREPA_ANT2:				INT;			(*calcul du temps nécessaire pour préparation des sources anticipées*)
	VAR_TPS_PREPA_ANT3:				INT;			(*calcul du temps nécessaire pour préparation des sources anticipées*)
	VAR_TPS_PREPA_ANT4:				INT;			(*calcul du temps nécessaire pour préparation des sources anticipées*)

	VAR_TPS_PREPA_ANT1_2s:			INT;			(*calcul du temps nécessaire pour préparation des sources anticipées en secondes + 2s*)
	VAR_TPS_PREPA_ANT2_2s:			INT;			(*calcul du temps nécessaire pour préparation des sources anticipées*)
	VAR_TPS_PREPA_ANT3_2s:			INT;			(*calcul du temps nécessaire pour préparation des sources anticipées*)
	VAR_TPS_PREPA_ANT4_2s:			INT;			(*calcul du temps nécessaire pour préparation des sources anticipées*)

	VAR_TPS_RESTANT_DEPOT:			INT;			(*temps restant en dépot calculé avec les épaisseurs et vitesses aggrégées, avec le PRM_Epaisseur*)
	VAR_CALCUL_VITESSE_THEORIQUE:	REAL;		(*vitesse aggrégée théorique*)

	TIMER_Lancement_Ant_S1:			TON;		(*timer de lancement de S1 anticipée*)
	TIMER_Lancement_Ant_S2:			TON;		(*timer de lancement de S2 anticipée*)
	TIMER_Lancement_Ant_S3:			TON;		(*timer de lancement de S3 anticipée*)
	TIMER_Lancement_Ant_S4:			TON;		(*timer de lancement de S4 anticipée*)

	FM_Prepa_Ant_S1:				R_TRIG;		(*Front montant de lancement de source 1 anticipée*)
	FM_Prepa_Ant_S2:				R_TRIG;		(*Front montant de lancement de source 2 anticipée*)
	FM_Prepa_Ant_S3:				R_TRIG;		(*Front montant de lancement de source 3 anticipée*)
	FM_Prepa_Ant_S4:				R_TRIG;		(*Front montant de lancement de source 4 anticipée*)

	VAR_Prepa_S1_Lancee:			BOOL;		(*indicateur de prépa S1 déja lancée*)
	VAR_Prepa_S2_Lancee:			BOOL;		(*indicateur de prépa S2 deja lancée*)
	VAR_Prepa_S3_Lancee:			BOOL;		(*indicateur de prépa S3 deja lancée*)
	VAR_Prepa_S4_Lancee:			BOOL;		(*indicateur de prépa S4 deja lancée*)

	VAR_Util_Gaz:					ARRAY[0..2] OF BOOL;		(*Indicateur des lignes de gaz utilisées*)
	VAR_Cond_MGaz:					BOOL;


	VAR_Cpt_Boucle:					USINT;		(*Compteur de boucle*)
	VAR_Step_To_Read:				USINT;		(*Indique le numéro de l'étape à lire*)
	VAR_Loop_In_Process:			BOOL;		(*Variable indiquant qu'une boucle est en cours d'execution*)

	TIMER_Stop_Controller:			TON;		(*timer de demande de stop du controleur de depot*)
	TIMER_Reset_Controller:			TON;		(*timer de demande de start du controleur de depot*)
END_VAR

	DEF_READ_LAYER.IdXML := '0';
	DEF_READ_LAYER.TagXML := 33;

	DEF_READ_LAYER_ANT.IdXML	:=	'0';
	DEF_READ_LAYER_ANT.TagXML	:=	33;

	EV_LOAD_LAYER.IdXML := '0';
	EV_LOAD_LAYER.TagXML :=34;
	EV_LOAD_LAYER.Groupe := 3;

	EV_NEXT_LAYER.IdXML :='0';
	EV_NEXT_LAYER.TagXML :=35;
	EV_NEXT_LAYER.Groupe := 3;
	
	EV_THICK_AGREGATE.IdXML := '0';
	EV_THICK_AGREGATE.TagXML := 43;
	EV_THICK_AGREGATE.Groupe := 3;

	DEF_RAZ_QZ.IDXML := '14';
	DEF_RAZ_QZ.TagXML :=5;

	DEF_QF.IDXML := '14';
	DEF_QF.TagXML :=9;

	DEF_PROG_QZ.IDXML := '14';
	DEF_PROG_QZ.TagXML :=4;

	DEF_CONTROLLER_STOPPED.IdXML := '14';
	DEF_CONTROLLER_STOPPED.TagXML := 17;

	EV_RELOAD.IdXML := '7';
	EV_RELOAD.TagXML := 15;
	EV_RELOAD.Groupe := 3;

	IdXML :='19';
	TagXML := 2;

IF  OP_RUN.AR THEN
	STATE_LAYER_TEXT := '';
END_IF

(*Reception des ordres*)
RQ_NEXT_LAYER := FALSE;
RCP_NEXT_LAYER:= M_NEXT_layer;


AUTOR_NEXT_LAYER	 :=	(OP_RUN.Etape.6 OR OP_RUN.Etape.7 OR OP_RUN.Etape.10
							OR OP_RUN.Etape.11 OR OP_RUN.Etape.12);

(*Evenement de lecture d'une couche*)
EV_LOAD_LAYER.VAL1 := UINT_TO_STRING(STATE_LAYER);
EV_LOAD_LAYER.VAL2 := STATE_LAYER_TEXT;
EV_LOAD_LAYER.CONDITION := OP_RUN.Etape.5 (*AND I_LAYER_LOADING_OK*);
EV_LOAD_LAYER();

EV_NEXT_LAYER.CONDITION := RCP_NEXT_LAYER AND AUTOR_NEXT_LAYER;
EV_NEXT_LAYER();

(*Evenement fin de couche*)
EV_THICK_AGREGATE.VAL1 := LREAL_TO_FMTSTR(REAL_TO_LREAL(STATE_THICKNESS_AGREGATE),3,TRUE);
EV_THICK_AGREGATE.CONDITION := STATE_END_OF_LAYER;
EV_THICK_AGREGATE();


RUN_PROCESS();

(*Temporisation de time out*)
TIMER_TIMEOUT	(
				PT:=T#5s,
				IN:=OP_RUN.Etape.4 OR OP_RUN.Etape.17
				);

(*Temporisation de time out de lecture de la couche anticipée*)
TIMER_TIMEOUT_ANT(
				PT := T#5s,
				IN := OP_RUN.Etape.5
				);

(*Demande de chargement procédé*)
RQ_READ_LAYER	:= 	OP_run.Etape.4;


(*Temporisation de time out de lecture de la couche anticipée*)
TIMER_Stop_Controller(
				PT := T#2s,
				IN := OP_RUN.Etape.2
				);


(*Temporisation de time out de lecture de la couche anticipée*)
TIMER_Reset_Controller(
				PT := T#2s,
				IN := OP_RUN.Etape.3
				);


(*Temporisation de time out de lecture de la couche anticipée*)
TIMER_RAZ_EPAISSEUR(
				PT := T#2s,
				IN := OP_RUN.Etape.11
				);

(*
(*Demande de chargement procédé sur le numéro d'étape de la boucle*)
RQ_READ_NUM_LAYER	:= OP_RUN.Etape.17;

(*Numéro de couche de départ de la boucle*)
OUT_NUM_LAYER_TO_READ	:= PRM_LOOP_FIRST_LAYER;
*)


(*Demande de lecture de la couche anticipée*)
RQ_READ_LAYER_ANT	:=	OP_RUN.Etape.5;


FM_ETAPE20(CLK:=OP_RUN.Etape.20);
FM_ETAPE6(CLK:=OP_RUN.Etape.6);
FM_ETAPE7(CLK:=OP_RUN.Etape.7);
FM_ETAPE9(CLK:=OP_RUN.Etape.9);
FM_ETAPE10(CLK:=OP_RUN.Etape.10);
FM_ETAPE11(CLK:=OP_RUN.Etape.11);
FM_ETAPE12(CLK:=OP_RUN.Etape.12);
FM_ETAPE13(CLK:=OP_RUN.Etape.13);
FM_ETAPE14(CLK:=OP_RUN.Etape.14);


IF NOT RQ_READ_LAYER THEN
	I_LAYER_LOADING_NOK := FALSE;
	I_LAYER_LOADING_OK:=FALSE;
	I_NO_MORE_LAYER :=FALSE;
END_IF

IF NOT RQ_READ_LAYER_ANT THEN
	I_LAYER_ANT_LOADING_NOK := FALSE;
	I_LAYER_ANT_LOADING_OK := FALSE;
	(*dans le cas de la couche anticipée, on ne remet pas le I_no_more_layer_ant à 0 ici*)
END_IF

(*remise à 0 du I_no_more_layer anticipée en étape 3, c'est à dire lors d'une nouvelle lecture de couche en cours*)
IF OP_RUN.Etape.4 THEN
	I_NO_MORE_LAYER_ANT := FALSE;
END_IF

(*Gestion du I_no_more_layer anticipée, on fait retomber les PRM_Util_sourceX_ant, ce qui inhibe toutes les actions*)
IF I_NO_MORE_LAYER_ANT THEN
	PRM_UTIL_SOURCE1_ANT := FALSE;
	PRM_UTIL_SOURCE2_ANT := FALSE;
	PRM_UTIL_SOURCE3_ANT := FALSE;
	PRM_UTIL_SOURCE4_ANT := FALSE;
END_IF


STATE_OK:=OP_RUN.OK;


(*Etat du grafcet d'empilement*)
STATUS	:= 	OP_RUN.STATUS;
(*Demande marche rotation PS*)
RQ_ROTATION_PS := FM_ETAPE6.Q AND NOT I_NO_ROTATION_PS;
(*Demande tilt PS*)
RQ_TILT_PS := FM_ETAPE7.Q;
(*Demande d'arrêt rotation PS*)
RQ_STOP_ROTATION_PS:= (FM_ETAPE6.Q AND I_NO_ROTATION_PS) OR FM_ETAPE14.Q;
(*Demande d'arrêt tilt PS*)
RQ_STOP_TILT_PS:=(FM_ETAPE6.Q AND I_MODE_TILT = 2) OR FM_ETAPE14.Q;
(*Demande marche chauffage*)
RQ_MARCHE_CHAUFFAGE := FM_ETAPE6.Q  AND (PRM_MODE_CHAUFFAGE = 1) AND CONF_CHAUFFAGE;
(*Demande arrêt chauffage*)
RQ_ARRET_CHAUFFAGE := FM_ETAPE6.Q  AND (PRM_MODE_CHAUFFAGE = 0) AND CONF_CHAUFFAGE;

(*Demande de positionnement du dôme à la position souhaitée pendant l'empilement.
	En fin d'empilement, positionnement du dôme en position haute*)
RQ_POSITIONNEMENT_Z := FM_ETAPE6.Q OR FM_ETAPE14.Q;

(*Consigne de position du dôme*)
(*IF RQ_POSITIONNEMENT_Z AND OP_RUN.Etape.14 THEN
	CONS_POSITION_DOME:= 1;
ELSIF RQ_POSITIONNEMENT_Z AND NOT OP_RUN.Etape.14 THEN
	CONS_POSITION_DOME:= PRM_Type_Dome +2;
END_IF*)

(*Demande marche IAD*)
RQ_MARCHE_IAD := FM_ETAPE7.Q AND  PRM_OP_UTIL_IAD AND CONF_IAD;
RQ_ARRET_IAD := (FM_ETAPE7.Q AND  NOT PRM_OP_UTIL_IAD) OR FM_Etape14.Q;

(*Demande ouverture cache IAD *)
RQ_OUV_CC_Iad := OP_RUN.Etape.12 AND PRM_OP_UTIL_IAD AND CONF_IAD;

(*Demande de chargement des parametres couches/quartz dans le contrôleur de dépôt*)
RQ_LOAD_PARAM:= OP_RUN.Etape.9;

(*Variable indiquant les lignes de gaz utilisées*)
VAR_Util_Gaz[1]:= (PRM_FLOW_GAZ1 > 0);
VAR_Util_Gaz[2]:= (PRM_FLOW_GAZ2 > 0);

(*Gestion présence gaz*)
(*MARCHE GAZ*)
IF OP_RUN.Etape.6 AND (PRM_N_SEGMENT_GAZ = 0) 	(*mise en gaz avant prefusion si gaz demandé dès le départ*)
	OR ( NOT OP_RUN.Etape.0 AND (PRM_N_SEGMENT_GAZ = 0) 		(*mise en gaz sur segments sélectionnés si gaz demandé dès le départ*)
		AND   (   	(PRM_UTIL_SOURCE1 AND PRM_GAZ_PRESSION_SEGMENT[I_N_SEGMENT_S1]) OR
				(PRM_UTIL_SOURCE2 AND PRM_GAZ_PRESSION_SEGMENT[I_N_SEGMENT_S2]) OR
				(PRM_UTIL_SOURCE3 AND PRM_GAZ_PRESSION_SEGMENT[I_N_SEGMENT_S3]) OR
				(PRM_UTIL_SOURCE4 AND PRM_GAZ_PRESSION_SEGMENT[I_N_SEGMENT_S4])	)	)
	OR ( NOT OP_RUN.Etape.0 AND NOT (PRM_N_SEGMENT_GAZ = 0) 	(*mise en gaz sur segments selectionnés et à partir du segement indiqué*)
		AND   (   	((I_N_SEGMENT_S1 >= PRM_N_SEGMENT_GAZ) AND PRM_UTIL_SOURCE1 AND PRM_GAZ_PRESSION_SEGMENT[I_N_SEGMENT_S1]) OR
				((I_N_SEGMENT_S2 >= PRM_N_SEGMENT_GAZ) AND PRM_UTIL_SOURCE2 AND PRM_GAZ_PRESSION_SEGMENT[I_N_SEGMENT_S2]) OR
				((I_N_SEGMENT_S3 >= PRM_N_SEGMENT_GAZ) AND PRM_UTIL_SOURCE3 AND PRM_GAZ_PRESSION_SEGMENT[I_N_SEGMENT_S3]) OR
				((I_N_SEGMENT_S4 >= PRM_N_SEGMENT_GAZ) AND PRM_UTIL_SOURCE4 AND PRM_GAZ_PRESSION_SEGMENT[I_N_SEGMENT_S4])	)	)
		THEN
			VAR_Cond_MGaz	:=	TRUE;
(*ARRET GAZ*)
ELSIF  ( NOT OP_RUN.Etape.0 AND (PRM_N_SEGMENT_GAZ = 0) 		(*arrêt gaz sur segments sélectionnés si gaz demandé dès le départ*)
		AND   (   	(PRM_UTIL_SOURCE1 AND NOT PRM_GAZ_PRESSION_SEGMENT[I_N_SEGMENT_S1]) OR
				(PRM_UTIL_SOURCE2 AND NOT PRM_GAZ_PRESSION_SEGMENT[I_N_SEGMENT_S2]) OR
				(PRM_UTIL_SOURCE3 AND NOT PRM_GAZ_PRESSION_SEGMENT[I_N_SEGMENT_S3]) OR
				(PRM_UTIL_SOURCE4 AND NOT PRM_GAZ_PRESSION_SEGMENT[I_N_SEGMENT_S4])	)	)
	OR ( NOT OP_RUN.Etape.0 AND NOT (PRM_N_SEGMENT_GAZ = 0) 	(*arrêt gaz sur segments selectionnés et à partir du segement indiqué*)
		AND   (   	((I_N_SEGMENT_S1 >= PRM_N_SEGMENT_GAZ) AND PRM_UTIL_SOURCE1 AND NOT PRM_GAZ_PRESSION_SEGMENT[I_N_SEGMENT_S1]) OR
				((I_N_SEGMENT_S2 >= PRM_N_SEGMENT_GAZ) AND PRM_UTIL_SOURCE2 AND NOT PRM_GAZ_PRESSION_SEGMENT[I_N_SEGMENT_S2]) OR
				((I_N_SEGMENT_S3 >= PRM_N_SEGMENT_GAZ) AND PRM_UTIL_SOURCE3 AND NOT PRM_GAZ_PRESSION_SEGMENT[I_N_SEGMENT_S3]) OR
				((I_N_SEGMENT_S4 >= PRM_N_SEGMENT_GAZ) AND PRM_UTIL_SOURCE4 AND NOT PRM_GAZ_PRESSION_SEGMENT[I_N_SEGMENT_S4])	)	)
	OR OP_RUN.Etape.14		(*fin empilement*)	
	OR OP_RUN.Etape.1
		THEN
			VAR_Cond_MGaz	:=	FALSE;

END_IF

FM_COND_MGAZ.CLK	:=	VAR_Cond_MGaz;
FM_COND_MGAZ();
FD_COND_MGAZ.CLK	:=	VAR_Cond_MGaz;
FD_COND_MGAZ();

(*Ordre de marche gaz*)
RQ_MARCHE_GAZ[1]  := FM_COND_MGAZ.Q AND VAR_Util_Gaz[1];
RQ_MARCHE_GAZ[2]  := FM_COND_MGAZ.Q AND VAR_Util_Gaz[2];

(*Demande arrêt des lignes de gaz*)
RQ_ARRET_GAZ[1] :=(FM_ETAPE6.Q AND NOT VAR_Util_Gaz[1]) OR FD_COND_MGAZ.Q;
RQ_ARRET_GAZ[2] :=(FM_ETAPE6.Q AND NOT VAR_Util_Gaz[2]) OR FD_COND_MGAZ.Q;

(*Demande marche régulation gaz ligne 1*)
RQ_MARCHE_REGUL_GAZ[1]:= FM_COND_MGAZ.Q AND (PRM_MODE_PUMPING = 2);
(*Demande arrêt régulation gaz ligne 1*)
RQ_ARRET_REGUL_GAZ[1]:= (FM_ETAPE13.Q AND (PRM_MODE_PUMPING = 2)) OR FD_COND_MGAZ.Q;

(*Demande de régulation gaz ligne 2*)
RQ_MARCHE_REGUL_GAZ[2]:= FM_COND_MGAZ.Q AND (PRM_MODE_PUMPING = 3);
(*Demande arrêt régulation gaz ligne 2*)
RQ_ARRET_REGUL_GAZ[2]:= (FM_ETAPE13.Q AND (PRM_MODE_PUMPING = 3)) OR FD_COND_MGAZ.Q;

(*Demande de mise en pompage procédé*)
RQ_MARCHE_POMPAGE_PROC:= FM_COND_MGAZ.Q AND (PRM_MODE_PUMPING = 0 OR PRM_MODE_PUMPING = 1);

(*Demande de mise en pompage secondaire*)
RQ_MARCHE_POMPAGE_SEC:=  FD_COND_MGAZ.Q;

